C01810=1192.674,149.566,-54.225,-178.267,6.243,148.616
C01811=1192.678,149.317,-54.204,-178.270,6.241,148.616
C01812=1192.683,149.068,-54.182,-178.272,6.240,148.617
C01813=1192.688,148.819,-54.161,-178.275,6.239,148.617
C01814=1192.693,148.570,-54.141,-178.278,6.237,148.618
C01815=1192.698,148.321,-54.119,-178.281,6.235,148.618
C01816=1192.701,148.072,-54.099,-178.283,6.234,148.618
C01817=1192.707,147.823,-54.078,-178.286,6.232,148.619
C01818=1192.712,147.573,-54.057,-178.289,6.231,148.619
C01819=1192.716,147.324,-54.036,-178.291,6.229,148.620
C01820=1192.721,147.076,-54.015,-178.294,6.228,148.620
C01821=1192.726,146.827,-53.994,-178.296,6.226,148.620
C01822=1192.731,146.577,-53.973,-178.299,6.225,148.621
C01823=1192.735,146.329,-53.953,-178.302,6.223,148.621
C01824=1192.740,146.079,-53.932,-178.304,6.222,148.622
C01825=1192.744,145.830,-53.911,-178.307,6.221,148.622
C01826=1192.749,145.581,-53.890,-178.310,6.219,148.623
C01827=1192.753,145.332,-53.869,-178.312,6.217,148.623
C01828=1192.759,145.083,-53.848,-178.315,6.216,148.624
C01829=1192.763,144.834,-53.828,-178.318,6.215,148.624
C01830=1192.768,144.585,-53.807,-178.320,6.213,148.624
C01831=1192.773,144.336,-53.787,-178.323,6.211,148.625
C01832=1192.778,144.086,-53.766,-178.325,6.211,148.625
C01833=1192.782,143.837,-53.745,-178.328,6.209,148.626
C01834=1192.787,143.588,-53.724,-178.331,6.207,148.626
C01835=1192.792,143.339,-53.704,-178.334,6.205,148.627
C01836=1192.797,143.091,-53.682,-178.336,6.204,148.627
C01837=1192.801,142.842,-53.662,-178.339,6.203,148.628
C01838=1192.806,142.592,-53.641,-178.342,6.201,148.628
C01839=1192.811,142.343,-53.620,-178.344,6.200,148.628
C01840=1192.815,142.093,-53.599,-178.346,6.198,148.629
C01841=1192.820,141.844,-53.579,-178.349,6.197,148.629
C01842=1192.824,141.596,-53.558,-178.352,6.195,148.630
C01843=1192.830,141.346,-53.538,-178.354,6.194,148.630
C01844=1192.834,141.097,-53.518,-178.357,6.192,148.630
C01845=1192.839,140.847,-53.497,-178.360,6.191,148.631
C01846=1192.844,140.598,-53.476,-178.362,6.190,148.632
C01847=1192.848,140.350,-53.456,-178.365,6.188,148.632
C01848=1192.853,140.100,-53.435,-178.368,6.187,148.632
C01849=1192.858,139.851,-53.415,-178.371,6.185,148.633
C01850=1192.862,139.602,-53.394,-178.373,6.184,148.633
C01851=1192.867,139.353,-53.373,-178.376,6.182,148.634
C01852=1192.872,139.104,-53.353,-178.378,6.181,148.634
C01853=1192.877,138.856,-53.333,-178.381,6.180,148.635
C01854=1192.882,138.606,-53.313,-178.384,6.178,148.635
C01855=1192.887,138.357,-53.292,-178.386,6.176,148.635
C01856=1192.891,138.108,-53.272,-178.388,6.176,148.636
C01857=1192.896,137.859,-53.251,-178.392,6.174,148.636
C01858=1192.901,137.610,-53.231,-178.394,6.172,148.637
C01859=1192.905,137.361,-53.210,-178.397,6.171,148.637
C01860=1192.911,137.111,-53.190,-178.399,6.170,148.638
C01861=1192.915,136.862,-53.170,-178.402,6.168,148.638
C01862=1192.920,136.613,-53.149,-178.405,6.166,148.639
C01863=1192.924,136.364,-53.129,-178.407,6.165,148.639
C01864=1192.930,136.114,-53.109,-178.410,6.164,148.639
C01865=1192.934,135.865,-53.088,-178.413,6.162,148.640
C01866=1192.938,135.616,-53.068,-178.415,6.161,148.640
C01867=1192.943,135.368,-53.048,-178.418,6.160,148.641
C01868=1192.949,135.118,-53.028,-178.420,6.158,148.641
C01869=1192.953,134.869,-53.007,-178.423,6.157,148.642
C01870=1192.958,134.620,-52.987,-178.426,6.155,148.642
C01871=1192.963,134.371,-52.967,-178.428,6.154,148.643
C01872=1192.967,134.122,-52.947,-178.431,6.153,148.643
C01873=1192.972,133.873,-52.926,-178.434,6.151,148.644
C01874=1192.977,133.623,-52.906,-178.436,6.150,148.644
C01875=1192.981,133.374,-52.886,-178.438,6.149,148.644
C01876=1192.987,133.105,-52.864,-178.442,6.147,148.645
C01877=1192.992,132.837,-52.842,-178.444,6.145,148.645
C01878=1192.997,132.568,-52.821,-178.448,6.144,148.646
C01879=1193.002,132.300,-52.799,-178.450,6.142,148.646
C01880=1193.007,132.051,-52.779,-178.453,6.142,148.647
C01881=1193.011,131.802,-52.759,-178.456,6.140,148.647
C01882=1193.017,131.552,-52.739,-178.458,6.138,148.648
C01883=1193.022,131.304,-52.719,-178.461,6.138,148.648
C01884=1193.026,131.054,-52.699,-178.464,6.136,148.649
C01885=1193.031,130.805,-52.679,-178.466,6.134,148.649
C01886=1193.036,130.555,-52.659,-178.468,6.133,148.650
C01887=1193.040,130.307,-52.639,-178.472,6.132,148.650
C01888=1193.045,130.058,-52.619,-178.474,6.130,148.651
C01889=1193.050,129.809,-52.599,-178.476,6.129,148.651
C01890=1193.055,129.559,-52.579,-178.479,6.128,148.652
C01891=1193.060,129.310,-52.558,-178.482,6.126,148.652
C01892=1193.064,129.060,-52.539,-178.484,6.125,148.652
C01893=1193.069,128.812,-52.519,-178.487,6.123,148.653
C01894=1193.074,128.562,-52.499,-178.490,6.123,148.653
C01895=1193.079,128.314,-52.479,-178.492,6.121,148.654
C01896=1193.083,128.064,-52.459,-178.495,6.119,148.655
C01897=1193.088,127.816,-52.439,-178.498,6.118,148.655
C01898=1193.093,127.566,-52.419,-178.500,6.117,148.655
C01899=1193.098,127.317,-52.400,-178.503,6.115,148.656
C01900=1193.102,127.068,-52.379,-178.506,6.114,148.656
C01901=1193.108,126.819,-52.360,-178.508,6.113,148.657
C01902=1193.112,126.569,-52.340,-178.510,6.112,148.657
C01903=1193.117,126.320,-52.320,-178.514,6.110,148.658
C01904=1193.122,126.071,-52.300,-178.516,6.108,148.658
C01905=1193.127,125.822,-52.281,-178.518,6.107,148.659
C01906=1193.131,125.573,-52.261,-178.522,6.106,148.659
C01907=1193.136,125.323,-52.241,-178.524,6.105,148.660
C01908=1193.141,125.074,-52.221,-178.526,6.103,148.660
C01909=1193.146,124.825,-52.201,-178.530,6.102,148.661
C01910=1193.150,124.576,-52.182,-178.532,6.101,148.661
C01911=1193.155,124.327,-52.163,-178.534,6.099,148.661
C01912=1193.159,124.077,-52.143,-178.538,6.098,148.662
C01913=1193.164,123.829,-52.123,-178.540,6.097,148.662
C01914=1193.169,123.579,-52.103,-178.542,6.095,148.663
C01915=1193.174,123.330,-52.084,-178.545,6.095,148.663
C01916=1193.179,123.081,-52.064,-178.548,6.093,148.664
C01917=1193.184,122.832,-52.044,-178.550,6.092,148.664
C01918=1193.188,122.582,-52.024,-178.553,6.090,148.665
C01919=1193.194,122.333,-52.005,-178.556,6.089,148.665
C01920=1193.198,122.084,-51.986,-178.558,6.088,148.666
C01921=1193.203,121.835,-51.966,-178.561,6.086,148.666
C01922=1193.208,121.586,-51.946,-178.563,6.085,148.667
C01923=1193.212,121.337,-51.927,-178.566,6.084,148.667
C01924=1193.217,121.087,-51.907,-178.569,6.082,148.668
C01925=1193.222,120.838,-51.888,-178.571,6.081,148.668
C01926=1193.227,120.589,-51.868,-178.574,6.080,148.669
C01927=1193.231,120.340,-51.849,-178.576,6.079,148.669
C01928=1193.237,120.091,-51.830,-178.579,6.077,148.670
C01929=1193.241,119.841,-51.810,-178.582,6.076,148.670
C01930=1193.246,119.592,-51.790,-178.584,6.075,148.671
C01931=1193.251,119.343,-51.770,-178.588,6.074,148.671
C01932=1193.255,119.094,-51.751,-178.590,6.073,148.672
C01933=1193.260,118.845,-51.732,-178.592,6.071,148.672
C01934=1193.265,118.596,-51.712,-178.595,6.070,148.673
C01935=1193.270,118.346,-51.693,-178.598,6.068,148.673
C01936=1193.274,118.097,-51.674,-178.600,6.068,148.673
C01937=1193.279,117.848,-51.654,-178.603,6.066,148.674
C01938=1193.285,117.599,-51.635,-178.606,6.064,148.674
C01939=1193.289,117.349,-51.615,-178.608,6.064,148.675
C01940=1193.293,117.100,-51.596,-178.611,6.062,148.676
C01941=1193.299,116.851,-51.577,-178.613,6.061,148.676
C01942=1193.303,116.602,-51.557,-178.616,6.060,148.677
C01943=1193.309,116.353,-51.538,-178.618,6.059,148.677
C01944=1193.313,116.104,-51.519,-178.621,6.057,148.677
C01945=1193.318,115.854,-51.500,-178.624,6.056,148.678
C01946=1193.323,115.605,-51.481,-178.627,6.055,148.678
C01947=1193.328,115.356,-51.462,-178.630,6.053,148.679
C01948=1193.333,115.106,-51.442,-178.632,6.052,148.679
C01949=1193.337,114.857,-51.423,-178.635,6.051,148.680
C01950=1193.342,114.608,-51.404,-178.637,6.050,148.681
C01951=1193.347,114.359,-51.384,-178.640,6.048,148.681
C01952=1193.352,114.110,-51.365,-178.642,6.048,148.682
C01953=1193.356,113.861,-51.346,-178.645,6.046,148.682
C01954=1193.362,113.611,-51.328,-178.647,6.045,148.682
C01955=1193.366,113.362,-51.308,-178.650,6.044,148.683
C01956=1193.371,113.113,-51.289,-178.653,6.043,148.683
C01957=1193.376,112.863,-51.270,-178.656,6.041,148.684
C01958=1193.381,112.615,-51.250,-178.658,6.040,148.684
C01959=1193.385,112.365,-51.232,-178.661,6.039,148.685
C01960=1193.391,112.116,-51.213,-178.664,6.037,148.685
C01961=1193.395,111.867,-51.194,-178.666,6.036,148.686
C01962=1193.400,111.618,-51.174,-178.669,6.035,148.687
C01963=1193.405,111.368,-51.155,-178.671,6.034,148.687
C01964=1193.410,111.119,-51.137,-178.674,6.032,148.687
C01965=1193.414,110.869,-51.117,-178.677,6.032,148.688
C01966=1193.419,110.621,-51.098,-178.679,6.030,148.688
C01967=1193.424,110.371,-51.079,-178.682,6.029,148.689
C01968=1193.429,110.122,-51.061,-178.685,6.028,148.689
C01969=1193.434,109.873,-51.041,-178.687,6.027,148.690
C01970=1193.438,109.624,-51.022,-178.690,6.025,148.690
C01971=1193.444,109.375,-51.004,-178.692,6.024,148.691
C01972=1193.448,109.125,-50.985,-178.695,6.023,148.691
C01973=1193.453,108.876,-50.965,-178.697,6.022,148.692
C01974=1193.457,108.627,-50.947,-178.700,6.021,148.693
C01975=1193.463,108.378,-50.928,-178.703,6.020,148.693
C01976=1193.467,108.128,-50.909,-178.706,6.018,148.694
C01977=1193.472,107.879,-50.890,-178.708,6.017,148.694
C01978=1193.477,107.630,-50.871,-178.711,6.016,148.694
C01979=1193.482,107.380,-50.852,-178.713,6.015,148.695
C01980=1193.488,107.112,-50.832,-178.716,6.013,148.695
C01981=1193.492,106.843,-50.812,-178.719,6.012,148.696
C01982=1193.498,106.575,-50.791,-178.722,6.011,148.697
C01983=1193.503,106.307,-50.772,-178.724,6.010,148.697
C01984=1193.507,106.057,-50.752,-178.727,6.009,148.698
C01985=1193.512,105.808,-50.734,-178.730,6.007,148.698
C01986=1193.518,105.559,-50.715,-178.732,6.007,148.699
C01987=1193.522,105.310,-50.697,-178.735,6.005,148.699
C01988=1193.527,105.061,-50.677,-178.738,6.004,148.700
C01989=1193.532,104.811,-50.659,-178.740,6.003,148.700
C01990=1193.536,104.562,-50.640,-178.743,6.002,148.701
C01991=1193.542,104.313,-50.622,-178.746,6.000,148.701
C01992=1193.546,104.064,-50.603,-178.748,5.999,148.702
C01993=1193.551,103.814,-50.584,-178.751,5.998,148.702
C01994=1193.556,103.565,-50.565,-178.753,5.997,148.703
C01995=1193.560,103.316,-50.547,-178.756,5.996,148.703
C01996=1193.566,103.066,-50.528,-178.759,5.995,148.704
C01997=1193.571,102.818,-50.510,-178.762,5.993,148.704
C01998=1193.575,102.568,-50.491,-178.764,5.992,148.705
C01999=1193.580,102.319,-50.472,-178.767,5.991,148.706
C02000=1193.585,102.070,-50.454,-178.769,5.990,148.706
C02001=1193.590,101.820,-50.436,-178.771,5.989,148.706
C02002=1193.595,101.571,-50.416,-178.774,5.988,148.707
C02003=1193.600,101.322,-50.398,-178.777,5.987,148.707
C02004=1193.604,101.072,-50.379,-178.780,5.985,148.708
C02005=1193.609,100.823,-50.361,-178.782,5.985,148.708
C02006=1193.614,100.574,-50.343,-178.785,5.983,148.709
C02007=1193.619,100.325,-50.324,-178.787,5.982,148.710
C02008=1193.623,100.075,-50.306,-178.790,5.981,148.710
C02009=1193.629,99.826,-50.287,-178.793,5.980,148.711
C02010=1193.634,99.577,-50.269,-178.796,5.979,148.711
C02011=1193.638,99.327,-50.250,-178.798,5.978,148.712
C02012=1193.643,99.078,-50.232,-178.801,5.977,148.712
C02013=1193.648,98.829,-50.214,-178.803,5.975,148.713
C02014=1193.653,98.580,-50.195,-178.806,5.975,148.713
C02015=1193.657,98.330,-50.177,-178.809,5.973,148.714
C02016=1193.662,98.081,-50.159,-178.811,5.972,148.714
C02017=1193.668,97.832,-50.140,-178.814,5.971,148.715
C02018=1193.673,97.583,-50.122,-178.816,5.970,148.715
C02019=1193.677,97.333,-50.103,-178.819,5.968,148.716
C02020=1193.682,97.084,-50.085,-178.821,5.967,148.716
C02021=1193.687,96.835,-50.067,-178.824,5.967,148.717
C02022=1193.692,96.585,-50.048,-178.827,5.965,148.717
C02023=1193.697,96.336,-50.030,-178.829,5.965,148.718
C02024=1193.701,96.087,-50.011,-178.832,5.963,148.718
C02025=1193.706,95.838,-49.993,-178.835,5.962,148.719
C02026=1193.711,95.589,-49.975,-178.837,5.961,148.719
C02027=1193.716,95.339,-49.957,-178.840,5.960,148.720
C02028=1193.720,95.090,-49.939,-178.842,5.959,148.721
C02029=1193.726,94.840,-49.921,-178.845,5.958,148.721
C02030=1193.731,94.591,-49.903,-178.847,5.957,148.722
C02031=1193.736,94.342,-49.885,-178.851,5.955,148.722
C02032=1193.741,94.093,-49.867,-178.853,5.954,148.723
C02033=1193.745,93.843,-49.848,-178.855,5.954,148.723
C02034=1193.750,93.594,-49.830,-178.858,5.952,148.724
C02035=1193.754,93.345,-49.812,-178.861,5.952,148.724
C02036=1193.759,93.096,-49.794,-178.863,5.950,148.725
C02037=1193.764,92.847,-49.776,-178.866,5.949,148.725
C02038=1193.770,92.597,-49.757,-178.868,5.948,148.726
C02039=1193.774,92.347,-49.739,-178.871,5.947,148.727
C02040=1193.779,92.098,-49.721,-178.874,5.946,148.727
C02041=1193.784,91.849,-49.703,-178.877,5.945,148.728
C02042=1193.789,91.600,-49.685,-178.879,5.944,148.728
C02043=1193.794,91.351,-49.667,-178.881,5.943,148.729
C02044=1193.799,91.101,-49.649,-178.884,5.941,148.729
C02045=1193.804,90.852,-49.631,-178.887,5.941,148.730
C02046=1193.808,90.602,-49.613,-178.890,5.939,148.730
C02047=1193.813,90.353,-49.595,-178.892,5.939,148.731
C02048=1193.818,90.104,-49.577,-178.895,5.938,148.731
C02049=1193.823,89.854,-49.559,-178.897,5.936,148.732
C02050=1193.828,89.605,-49.541,-178.900,5.936,148.732
C02051=1193.833,89.356,-49.523,-178.903,5.934,148.733
C02052=1193.838,89.107,-49.505,-178.905,5.933,148.734
C02053=1193.843,88.857,-49.487,-178.908,5.933,148.734
C02054=1193.848,88.608,-49.469,-178.911,5.931,148.735
C02055=1193.852,88.358,-49.451,-178.913,5.930,148.735
C02056=1193.857,88.109,-49.433,-178.916,5.930,148.736
C02057=1193.862,87.859,-49.416,-178.918,5.928,148.736
C02058=1193.867,87.610,-49.398,-178.921,5.927,148.737
C02059=1193.872,87.361,-49.380,-178.924,5.926,148.737
C02060=1193.877,87.112,-49.362,-178.926,5.925,148.738
C02061=1193.882,86.863,-49.344,-178.928,5.924,148.738
C02062=1193.886,86.614,-49.326,-178.932,5.923,148.739
C02063=1193.891,86.364,-49.309,-178.934,5.922,148.739
C02064=1193.896,86.115,-49.291,-178.936,5.921,148.740
C02065=1193.901,85.866,-49.273,-178.939,5.920,148.741
C02066=1193.906,85.617,-49.255,-178.942,5.919,148.741
C02067=1193.911,85.367,-49.238,-178.945,5.918,148.742
C02068=1193.916,85.118,-49.220,-178.947,5.917,148.742
C02069=1193.921,84.868,-49.202,-178.950,5.916,148.743
C02070=1193.926,84.619,-49.184,-178.952,5.915,148.743
C02071=1193.930,84.370,-49.167,-178.955,5.914,148.744
C02072=1193.935,84.121,-49.149,-178.957,5.913,148.744
C02073=1193.940,83.871,-49.131,-178.960,5.912,148.745
C02074=1193.945,83.622,-49.114,-178.962,5.911,148.745
C02075=1193.950,83.372,-49.096,-178.965,5.910,148.746
C02076=1193.955,83.123,-49.078,-178.968,5.909,148.747
C02077=1193.960,82.874,-49.062,-178.970,5.908,148.747
C02078=1193.965,82.625,-49.044,-178.973,5.907,148.748
C02079=1193.969,82.375,-49.026,-178.976,5.906,148.748
C02080=1193.975,82.126,-49.008,-178.978,5.905,148.749
C02081=1193.980,81.876,-48.990,-178.980,5.904,148.749
C02082=1193.984,81.628,-48.973,-178.984,5.903,148.750
C02083=1193.989,81.378,-48.956,-178.986,5.902,148.750
C02084=1193.994,81.110,-48.936,-178.989,5.901,148.751
C02085=1193.999,80.841,-48.918,-178.992,5.900,148.752
C02086=1194.005,80.572,-48.898,-178.995,5.899,148.752
C02087=1194.010,80.304,-48.880,-178.997,5.898,148.753
C02088=1194.015,80.055,-48.862,-179.000,5.897,148.753
C02089=1194.020,79.806,-48.845,-179.003,5.896,148.754
C02090=1194.025,79.556,-48.827,-179.005,5.895,148.754
C02091=1194.030,79.307,-48.810,-179.008,5.894,148.755
C02092=1194.034,79.058,-48.793,-179.010,5.893,148.755
C02093=1194.039,78.808,-48.775,-179.013,5.892,148.756
C02094=1194.044,78.559,-48.757,-179.015,5.891,148.757
C02095=1194.050,78.309,-48.740,-179.018,5.890,148.757
C02096=1194.054,78.060,-48.723,-179.021,5.889,148.758
C02097=1194.059,77.810,-48.705,-179.023,5.888,148.758
C02098=1194.064,77.561,-48.687,-179.026,5.887,148.759
C02099=1194.068,77.312,-48.671,-179.028,5.886,148.759
C02100=1194.074,77.063,-48.653,-179.031,5.885,148.760
C02101=1194.079,76.813,-48.636,-179.034,5.884,148.760
C02102=1194.084,76.564,-48.619,-179.036,5.883,148.761
C02103=1194.088,76.315,-48.601,-179.039,5.883,148.762
C02104=1194.094,76.065,-48.584,-179.042,5.881,148.762
C02105=1194.098,75.816,-48.567,-179.044,5.880,148.763
C02106=1194.103,75.566,-48.549,-179.046,5.879,148.763
C02107=1194.108,75.317,-48.533,-179.049,5.879,148.764
C02108=1194.112,75.068,-48.515,-179.052,5.878,148.765
C02109=1194.118,74.819,-48.498,-179.054,5.877,148.765
C02110=1194.123,74.569,-48.481,-179.057,5.876,148.766
C02111=1194.128,74.320,-48.463,-179.060,5.874,148.766
C02112=1194.133,74.070,-48.446,-179.062,5.874,148.767
C02113=1194.137,73.821,-48.429,-179.065,5.873,148.767
C02114=1194.142,73.571,-48.411,-179.068,5.872,148.768
C02115=1194.147,73.323,-48.395,-179.070,5.871,148.769
C02116=1194.153,73.073,-48.378,-179.073,5.870,148.769
C02117=1194.157,72.824,-48.360,-179.075,5.870,148.770
C02118=1194.162,72.574,-48.343,-179.078,5.868,148.770
C02119=1194.166,72.325,-48.326,-179.080,5.867,148.771
C02120=1194.172,72.075,-48.309,-179.083,5.867,148.771
C02121=1194.177,71.826,-48.291,-179.085,5.866,148.772
C02122=1194.182,71.577,-48.275,-179.088,5.864,148.772
C02123=1194.187,71.327,-48.258,-179.091,5.864,148.773
C02124=1194.191,71.078,-48.241,-179.093,5.863,148.774
C02125=1194.196,70.828,-48.223,-179.096,5.862,148.774
C02126=1194.201,70.580,-48.207,-179.099,5.861,148.775
C02127=1194.207,70.330,-48.189,-179.101,5.860,148.775
C02128=1194.211,70.080,-48.173,-179.104,5.860,148.776
C02129=1194.216,69.831,-48.155,-179.107,5.858,148.776
C02130=1194.220,69.582,-48.138,-179.109,5.857,148.777
C02131=1194.226,69.333,-48.121,-179.111,5.856,148.777
C02132=1194.231,69.083,-48.104,-179.114,5.856,148.778
C02133=1194.236,68.833,-48.087,-179.117,5.855,148.779
C02134=1194.240,68.584,-48.071,-179.119,5.854,148.779
C02135=1194.246,68.335,-48.054,-179.122,5.853,148.780
C02136=1194.251,68.085,-48.037,-179.125,5.851,148.780
C02137=1194.255,67.836,-48.020,-179.127,5.851,148.781
C02138=1194.260,67.587,-48.002,-179.130,5.850,148.782
C02139=1194.265,67.338,-47.986,-179.132,5.849,148.782
C02140=1194.270,67.088,-47.969,-179.135,5.848,148.783
C02141=1194.275,66.839,-47.952,-179.138,5.848,148.783
C02142=1194.279,66.589,-47.935,-179.140,5.847,148.784
C02143=1194.285,66.340,-47.918,-179.143,5.846,148.784
C02144=1194.290,66.091,-47.902,-179.145,5.844,148.785
C02145=1194.295,65.841,-47.885,-179.148,5.844,148.786
C02146=1194.300,65.592,-47.868,-179.151,5.843,148.786
C02147=1194.304,65.342,-47.852,-179.153,5.842,148.787
C02148=1194.310,65.093,-47.834,-179.156,5.841,148.787
C02149=1194.314,64.843,-47.818,-179.159,5.840,148.788
C02150=1194.319,64.594,-47.801,-179.161,5.840,148.788
C02151=1194.324,64.345,-47.784,-179.163,5.839,148.789
C02152=1194.329,64.095,-47.767,-179.166,5.838,148.790
C02153=1194.334,63.846,-47.751,-179.169,5.837,148.790
C02154=1194.339,63.597,-47.734,-179.171,5.836,148.791
C02155=1194.344,63.347,-47.717,-179.174,5.835,148.791
C02156=1194.349,63.098,-47.701,-179.176,5.835,148.792
C02157=1194.354,62.848,-47.684,-179.179,5.833,148.793
C02158=1194.358,62.599,-47.667,-179.182,5.833,148.793
C02159=1194.364,62.350,-47.651,-179.184,5.832,148.794
C02160=1194.369,62.100,-47.634,-179.186,5.831,148.794
C02161=1194.374,61.850,-47.617,-179.190,5.830,148.795
C02162=1194.379,61.602,-47.601,-179.192,5.829,148.795
C02163=1194.383,61.352,-47.584,-179.194,5.828,148.796
C02164=1194.388,61.102,-47.567,-179.197,5.828,148.797
C02165=1194.393,60.853,-47.551,-179.200,5.827,148.797
C02166=1194.398,60.604,-47.534,-179.202,5.826,148.798
C02167=1194.403,60.355,-47.519,-179.205,5.825,148.798
C02168=1194.409,60.105,-47.501,-179.208,5.824,148.799
C02169=1194.413,59.855,-47.485,-179.210,5.824,148.799
C02170=1194.418,59.607,-47.468,-179.212,5.823,148.800
C02171=1194.423,59.357,-47.452,-179.216,5.822,148.801
C02172=1194.429,59.107,-47.436,-179.218,5.821,148.801
C02173=1194.433,58.858,-47.419,-179.220,5.820,148.802
C02174=1194.438,58.608,-47.402,-179.223,5.820,148.802
C02175=1194.443,58.360,-47.386,-179.225,5.819,148.803
C02176=1194.448,58.109,-47.370,-179.228,5.817,148.804
C02177=1194.453,57.860,-47.353,-179.231,5.817,148.804
C02178=1194.458,57.611,-47.336,-179.233,5.816,148.805
C02179=1194.462,57.361,-47.320,-179.236,5.815,148.805
C02180=1194.468,57.112,-47.304,-179.238,5.815,148.806
C02181=1194.472,56.863,-47.287,-179.241,5.813,148.806
C02182=1194.477,56.614,-47.271,-179.244,5.813,148.807
C02183=1194.483,56.363,-47.255,-179.246,5.812,148.808
C02184=1194.488,56.115,-47.238,-179.249,5.811,148.808
C02185=1194.492,55.865,-47.222,-179.251,5.811,148.809
C02186=1194.498,55.616,-47.206,-179.254,5.809,148.809
C02187=1194.502,55.366,-47.189,-179.257,5.809,148.810
C02188=1194.508,55.098,-47.172,-179.259,5.808,148.811
C02189=1194.512,54.829,-47.154,-179.262,5.807,148.811
C02190=1194.519,54.560,-47.137,-179.265,5.806,148.812
C02191=1194.524,54.292,-47.119,-179.268,5.806,148.813
C02192=1194.529,54.042,-47.103,-179.270,5.805,148.813
C02193=1194.534,53.794,-47.087,-179.273,5.803,148.814
C02194=1194.538,53.544,-47.070,-179.276,5.803,148.814
C02195=1194.544,53.295,-47.054,-179.278,5.802,148.815
C02196=1194.548,53.045,-47.038,-179.280,5.801,148.816
C02197=1194.554,52.796,-47.022,-179.283,5.801,148.816
C02198=1194.558,52.546,-47.005,-179.285,5.800,148.817
C02199=1194.563,52.297,-46.990,-179.288,5.799,148.817
C02200=1194.568,52.047,-46.973,-179.291,5.798,148.818
C02201=1194.573,51.798,-46.958,-179.293,5.797,148.818
C02202=1194.578,51.549,-46.941,-179.296,5.797,148.819
C02203=1194.583,51.299,-46.925,-179.299,5.796,148.820
C02204=1194.588,51.050,-46.909,-179.301,5.795,148.820
C02205=1194.593,50.800,-46.893,-179.304,5.794,148.821
C02206=1194.597,50.551,-46.876,-179.307,5.793,148.822
C02207=1194.603,50.301,-46.861,-179.309,5.792,148.822
C02208=1194.607,50.052,-46.844,-179.311,5.792,148.823
C02209=1194.613,49.803,-46.829,-179.314,5.791,148.823
C02210=1194.617,49.553,-46.812,-179.316,5.791,148.824
C02211=1194.623,49.304,-46.796,-179.319,5.789,148.824
C02212=1194.628,49.055,-46.780,-179.322,5.789,148.825
C02213=1194.632,48.805,-46.764,-179.324,5.788,148.826
C02214=1194.638,48.555,-46.748,-179.327,5.787,148.826
C02215=1194.642,48.306,-46.732,-179.329,5.787,148.827
C02216=1194.648,48.056,-46.716,-179.332,5.786,148.827
C02217=1194.652,47.807,-46.700,-179.334,5.785,148.828
C02218=1194.658,47.558,-46.684,-179.337,5.784,148.829
C02219=1194.663,47.308,-46.668,-179.340,5.783,148.829
C02220=1194.667,47.059,-46.652,-179.342,5.783,148.830
C02221=1194.673,46.809,-46.636,-179.345,5.782,148.830
C02222=1194.678,46.559,-46.620,-179.347,5.781,148.831
C02223=1194.683,46.310,-46.604,-179.350,5.781,148.832
C02224=1194.687,46.061,-46.589,-179.352,5.780,148.832
C02225=1194.692,45.811,-46.573,-179.355,5.779,148.833
C02226=1194.697,45.562,-46.557,-179.358,5.778,148.833
C02227=1194.702,45.312,-46.541,-179.360,5.777,148.834
C02228=1194.707,45.063,-46.525,-179.363,5.777,148.835
C02229=1194.712,44.814,-46.509,-179.366,5.776,148.835
C02230=1194.717,44.564,-46.493,-179.368,5.775,148.836
C02231=1194.723,44.315,-46.477,-179.370,5.775,148.836
C02232=1194.727,44.066,-46.462,-179.373,5.774,148.837
C02233=1194.732,43.816,-46.446,-179.376,5.773,148.838
C02234=1194.737,43.567,-46.430,-179.378,5.772,148.838
C02235=1194.742,43.317,-46.414,-179.381,5.772,148.839
C02236=1194.747,43.067,-46.398,-179.383,5.771,148.839
C02237=1194.753,42.818,-46.383,-179.386,5.770,148.840
C02238=1194.756,42.569,-46.367,-179.388,5.770,148.841
C02239=1194.762,42.319,-46.351,-179.391,5.769,148.841
C02240=1194.767,42.070,-46.336,-179.393,5.768,148.842
C02241=1194.773,41.820,-46.320,-179.396,5.768,148.842
C02242=1194.777,41.570,-46.304,-179.399,5.766,148.843
C02243=1194.782,41.322,-46.288,-179.401,5.766,148.844
C02244=1194.787,41.072,-46.273,-179.404,5.765,148.844
C02245=1194.792,40.822,-46.257,-179.407,5.764,148.845
C02246=1194.797,40.573,-46.241,-179.409,5.764,148.845
C02247=1194.802,40.324,-46.226,-179.411,5.763,148.846
C02248=1194.807,40.074,-46.210,-179.414,5.763,148.847
C02249=1194.812,39.824,-46.195,-179.417,5.762,148.847
C02250=1194.818,39.575,-46.179,-179.419,5.761,148.848
C02251=1194.822,39.326,-46.164,-179.422,5.760,148.849
C02252=1194.827,39.076,-46.147,-179.425,5.759,148.849
C02253=1194.832,38.827,-46.132,-179.427,5.758,148.850
C02254=1194.837,38.577,-46.116,-179.429,5.758,148.850
C02255=1194.841,38.328,-46.101,-179.432,5.757,148.851
C02256=1194.847,38.078,-46.085,-179.435,5.757,148.852
C02257=1194.852,37.829,-46.070,-179.437,5.756,148.852
C02258=1194.857,37.580,-46.055,-179.439,5.755,148.853
C02259=1194.862,37.330,-46.039,-179.442,5.755,148.853
C02260=1194.867,37.080,-46.023,-179.445,5.754,148.854
C02261=1194.872,36.831,-46.008,-179.447,5.754,148.855
C02262=1194.877,36.582,-45.993,-179.450,5.752,148.855
C02263=1194.882,36.332,-45.977,-179.453,5.752,148.856
C02264=1194.887,36.083,-45.962,-179.455,5.751,148.856
C02265=1194.892,35.833,-45.946,-179.458,5.750,148.857
C02266=1194.897,35.584,-45.930,-179.460,5.750,148.858
C02267=1194.902,35.335,-45.915,-179.463,5.749,148.858
C02268=1194.907,35.085,-45.900,-179.465,5.748,148.859
C02269=1194.912,34.835,-45.884,-179.468,5.748,148.860
C02270=1194.917,34.585,-45.870,-179.470,5.747,148.860
C02271=1194.922,34.336,-45.854,-179.472,5.746,148.861
C02272=1194.927,34.087,-45.839,-179.475,5.746,148.861
C02273=1194.932,33.837,-45.823,-179.478,5.745,148.862
C02274=1194.937,33.587,-45.808,-179.480,5.745,148.863
C02275=1194.942,33.338,-45.793,-179.483,5.744,148.863
C02276=1194.947,33.089,-45.777,-179.486,5.743,148.864
C02277=1194.952,32.840,-45.762,-179.488,5.742,148.864
C02278=1194.957,32.590,-45.746,-179.491,5.742,148.865
C02279=1194.962,32.340,-45.732,-179.493,5.741,148.866
C02280=1194.967,32.091,-45.716,-179.496,5.740,148.866
C02281=1194.972,31.842,-45.701,-179.499,5.740,148.867
C02282=1194.977,31.592,-45.686,-179.501,5.739,148.868
C02283=1194.983,31.343,-45.670,-179.503,5.738,148.868
C02284=1194.987,31.093,-45.655,-179.506,5.738,148.869
C02285=1194.992,30.843,-45.640,-179.509,5.737,148.869
C02286=1194.997,30.594,-45.625,-179.511,5.736,148.870
C02287=1195.002,30.344,-45.609,-179.513,5.736,148.871
C02288=1195.007,30.095,-45.594,-179.516,5.735,148.871
C02289=1195.013,29.845,-45.579,-179.519,5.735,148.872
C02290=1195.017,29.596,-45.564,-179.521,5.734,148.872
C02291=1195.022,29.346,-45.548,-179.523,5.734,148.873
C02292=1195.027,29.077,-45.533,-179.527,5.732,148.874
C02293=1195.033,28.809,-45.516,-179.529,5.732,148.874
C02294=1195.038,28.540,-45.500,-179.532,5.731,148.875
C02295=1195.044,28.271,-45.484,-179.535,5.731,148.876
C02296=1195.048,28.022,-45.469,-179.537,5.730,148.876
C02297=1195.054,27.773,-45.453,-179.539,5.729,148.877
C02298=1195.059,27.523,-45.439,-179.542,5.729,148.878
C02299=1195.064,27.273,-45.423,-179.545,5.728,148.878
C02300=1195.069,27.024,-45.408,-179.547,5.728,148.879
C02301=1195.074,26.775,-45.394,-179.550,5.727,148.879
C02302=1195.079,26.525,-45.378,-179.552,5.726,148.880
C02303=1195.084,26.276,-45.363,-179.555,5.726,148.881
C02304=1195.089,26.026,-45.348,-179.557,5.725,148.881
C02305=1195.094,25.776,-45.333,-179.560,5.725,148.882
C02306=1195.099,25.527,-45.318,-179.563,5.723,148.883
C02307=1195.104,25.277,-45.303,-179.566,5.723,148.883
C02308=1195.109,25.028,-45.288,-179.568,5.722,148.884
C02309=1195.114,24.778,-45.273,-179.570,5.721,148.884
C02310=1195.119,24.529,-45.258,-179.573,5.721,148.885
C02311=1195.124,24.279,-45.244,-179.576,5.720,148.886
C02312=1195.129,24.030,-45.229,-179.578,5.720,148.886
C02313=1195.134,23.781,-45.214,-179.580,5.719,148.887
C02314=1195.139,23.531,-45.199,-179.583,5.718,148.888
C02315=1195.144,23.282,-45.184,-179.586,5.718,148.888
C02316=1195.149,23.032,-45.169,-179.588,5.717,148.889
C02317=1195.154,22.783,-45.154,-179.591,5.717,148.889
C02318=1195.160,22.533,-45.140,-179.593,5.716,148.890
C02319=1195.164,22.284,-45.125,-179.596,5.715,148.891
C02320=1195.169,22.034,-45.110,-179.598,5.715,148.891
C02321=1195.174,21.785,-45.095,-179.601,5.714,148.892
C02322=1195.179,21.535,-45.080,-179.603,5.714,148.892
C02323=1195.184,21.286,-45.065,-179.606,5.713,148.893
C02324=1195.190,21.036,-45.051,-179.609,5.713,148.894
C02325=1195.194,20.787,-45.036,-179.611,5.712,148.895
C02326=1195.199,20.537,-45.021,-179.613,5.711,148.895
C02327=1195.205,20.288,-45.006,-179.616,5.711,148.896
C02328=1195.210,20.038,-44.991,-179.619,5.710,148.896
C02329=1195.215,19.788,-44.977,-179.621,5.710,148.897
C02330=1195.219,19.539,-44.962,-179.623,5.709,148.897
C02331=1195.225,19.289,-44.947,-179.626,5.708,148.898
C02332=1195.230,19.040,-44.932,-179.629,5.708,148.899
C02333=1195.235,18.790,-44.918,-179.631,5.707,148.900
C02334=1195.240,18.541,-44.904,-179.634,5.706,148.900
C02335=1195.244,18.291,-44.889,-179.636,5.706,148.901
C02336=1195.250,18.041,-44.874,-179.639,5.705,148.901
C02337=1195.255,17.792,-44.860,-179.642,5.705,148.902
C02338=1195.260,17.543,-44.845,-179.644,5.704,148.902
C02339=1195.264,17.293,-44.830,-179.646,5.704,148.903
C02340=1195.270,17.043,-44.815,-179.649,5.703,148.904
C02341=1195.275,16.794,-44.800,-179.652,5.703,148.905
C02342=1195.280,16.545,-44.787,-179.654,5.702,148.905
C02343=1195.285,16.295,-44.772,-179.656,5.701,148.906
C02344=1195.290,16.046,-44.757,-179.659,5.701,148.906
C02345=1195.295,15.796,-44.743,-179.662,5.700,148.907
C02346=1195.301,15.546,-44.728,-179.664,5.700,148.908
C02347=1195.305,15.297,-44.713,-179.667,5.699,148.908
C02348=1195.310,15.047,-44.699,-179.669,5.699,148.909
C02349=1195.315,14.798,-44.685,-179.671,5.699,148.910
C02350=1195.320,14.548,-44.670,-179.674,5.698,148.910
C02351=1195.325,14.299,-44.655,-179.677,5.698,148.911
C02352=1195.330,14.050,-44.641,-179.679,5.697,148.911
C02353=1195.336,13.800,-44.626,-179.681,5.696,148.912
C02354=1195.341,13.550,-44.612,-179.684,5.696,148.913
C02355=1195.346,13.301,-44.598,-179.687,5.695,148.913
C02356=1195.351,13.051,-44.583,-179.689,5.694,148.914
C02357=1195.356,12.802,-44.569,-179.691,5.694,148.915
C02358=1195.361,12.552,-44.554,-179.694,5.693,148.915
C02359=1195.365,12.302,-44.540,-179.697,5.693,148.916
C02360=1195.371,12.053,-44.526,-179.699,5.692,148.916
C02361=1195.376,11.804,-44.512,-179.702,5.692,148.917
C02362=1195.381,11.554,-44.497,-179.704,5.691,148.918
C02363=1195.386,11.305,-44.483,-179.707,5.691,148.918
C02364=1195.391,11.055,-44.468,-179.710,5.690,148.919
C02365=1195.396,10.805,-44.453,-179.712,5.689,148.920
C02366=1195.401,10.555,-44.439,-179.714,5.689,148.920
C02367=1195.407,10.306,-44.425,-179.717,5.688,148.921
C02368=1195.412,10.057,-44.411,-179.720,5.688,148.922
C02369=1195.417,9.807,-44.397,-179.722,5.687,148.922
C02370=1195.421,9.558,-44.382,-179.724,5.686,148.923
C02371=1195.426,9.308,-44.367,-179.727,5.686,148.923
C02372=1195.432,9.059,-44.354,-179.729,5.686,148.924
C02373=1195.437,8.809,-44.339,-179.732,5.686,148.925
C02374=1195.442,8.560,-44.325,-179.734,5.685,148.925
C02375=1195.447,8.310,-44.311,-179.737,5.684,148.926
C02376=1195.452,8.060,-44.296,-179.739,5.684,148.927
C02377=1195.457,7.811,-44.283,-179.742,5.683,148.927
C02378=1195.462,7.562,-44.268,-179.745,5.683,148.928
C02379=1195.467,7.312,-44.254,-179.747,5.682,148.928
C02380=1195.472,7.062,-44.240,-179.749,5.681,148.929
C02381=1195.477,6.812,-44.225,-179.752,5.681,148.930
C02382=1195.483,6.563,-44.212,-179.755,5.681,148.931
C02383=1195.488,6.314,-44.197,-179.757,5.680,148.931
C02384=1195.492,6.064,-44.184,-179.760,5.679,148.932
C02385=1195.497,5.815,-44.169,-179.762,5.679,148.932
C02386=1195.502,5.566,-44.155,-179.765,5.678,148.933
C02387=1195.507,5.316,-44.141,-179.767,5.678,148.934
C02388=1195.512,5.066,-44.127,-179.769,5.678,148.934
C02389=1195.517,4.816,-44.113,-179.772,5.677,148.935
C02390=1195.523,4.567,-44.099,-179.774,5.677,148.936
C02391=1195.528,4.317,-44.085,-179.777,5.676,148.936
C02392=1195.533,4.067,-44.071,-179.780,5.676,148.937
C02393=1195.538,3.818,-44.057,-179.782,5.675,148.937
C02394=1195.543,3.569,-44.043,-179.785,5.674,148.938
C02395=1195.548,3.319,-44.029,-179.787,5.674,148.939
C02396=1195.553,3.050,-44.014,-179.790,5.673,148.939
C02397=1195.558,2.780,-43.999,-179.792,5.673,148.940
C02398=1195.564,2.512,-43.983,-179.795,5.672,148.941
C02399=1195.570,2.243,-43.969,-179.798,5.672,148.942
C02400=1195.575,1.993,-43.954,-179.800,5.671,148.942
C02401=1195.580,1.743,-43.940,-179.803,5.671,148.943
C02402=1195.585,1.494,-43.927,-179.805,5.670,148.943
C02403=1195.590,1.244,-43.913,-179.808,5.670,148.944
C02404=1195.595,0.994,-43.898,-179.811,5.669,148.945
C02405=1195.600,0.745,-43.885,-179.813,5.669,148.945
C02406=1195.605,0.496,-43.871,-179.815,5.669,148.946
C02407=1195.610,0.246,-43.857,-179.817,5.668,148.947
C02408=1195.615,-0.004,-43.843,-179.820,5.668,148.947
C02409=1195.621,-0.253,-43.829,-179.823,5.667,148.948
C02410=1195.625,-0.502,-43.815,-179.825,5.667,148.949
C02411=1195.630,-0.753,-43.802,-179.828,5.666,148.949
C02412=1195.636,-1.002,-43.788,-179.830,5.665,148.950
C02413=1195.641,-1.251,-43.774,-179.833,5.665,148.950
C02414=1195.646,-1.500,-43.760,-179.836,5.664,148.951
C02415=1195.651,-1.750,-43.747,-179.838,5.664,148.952
C02416=1195.656,-2.000,-43.732,-179.840,5.664,148.952
C02417=1195.661,-2.249,-43.718,-179.842,5.663,148.953
C02418=1195.667,-2.500,-43.705,-179.845,5.663,148.954
C02419=1195.671,-2.749,-43.691,-179.848,5.662,148.954
C02420=1195.676,-2.998,-43.677,-179.850,5.662,148.955
C02421=1195.682,-3.248,-43.664,-179.853,5.661,148.956
C02422=1195.687,-3.498,-43.649,-179.855,5.660,148.956
C02423=1195.692,-3.747,-43.636,-179.858,5.660,148.957
C02424=1195.697,-3.997,-43.623,-179.861,5.659,148.958
C02425=1195.702,-4.246,-43.609,-179.863,5.660,148.958
C02426=1195.707,-4.495,-43.595,-179.865,5.659,148.959
C02427=1195.712,-4.746,-43.581,-179.867,5.658,148.959
C02428=1195.717,-4.995,-43.568,-179.870,5.658,148.960
C02429=1195.722,-5.245,-43.555,-179.873,5.657,148.961
C02430=1195.727,-5.494,-43.541,-179.875,5.657,148.962
C02431=1195.732,-5.744,-43.526,-179.878,5.656,148.962
C02432=1195.737,-5.994,-43.513,-179.880,5.656,148.963
C02433=1195.742,-6.243,-43.500,-179.882,5.656,148.963
C02434=1195.748,-6.493,-43.486,-179.885,5.656,148.964
C02435=1195.753,-6.742,-43.473,-179.888,5.655,148.965
C02436=1195.758,-6.992,-43.459,-179.890,5.654,148.965
C02437=1195.763,-7.241,-43.445,-179.892,5.654,148.966
C02438=1195.768,-7.490,-43.431,-179.895,5.653,148.967
C02439=1195.773,-7.741,-43.418,-179.898,5.653,148.967
C02440=1195.778,-7.990,-43.404,-179.900,5.653,148.968
C02441=1195.783,-8.240,-43.391,-179.902,5.653,148.969
C02442=1195.788,-8.489,-43.377,-179.905,5.652,148.969
C02443=1195.793,-8.739,-43.364,-179.907,5.651,148.970
C02444=1195.799,-8.988,-43.350,-179.910,5.651,148.971
C02445=1195.804,-9.238,-43.337,-179.913,5.650,148.971
C02446=1195.809,-9.487,-43.323,-179.915,5.650,148.972
C02447=1195.814,-9.737,-43.310,-179.917,5.650,148.972
C02448=1195.819,-9.986,-43.297,-179.920,5.649,148.973
C02449=1195.824,-10.236,-43.283,-179.922,5.649,148.974
C02450=1195.828,-10.486,-43.270,-179.925,5.648,148.974
C02451=1195.834,-10.735,-43.256,-179.927,5.648,148.975
C02452=1195.839,-10.985,-43.242,-179.930,5.647,148.976
C02453=1195.844,-11.234,-43.229,-179.932,5.647,148.976
C02454=1195.849,-11.484,-43.216,-179.934,5.647,148.977
C02455=1195.855,-11.734,-43.203,-179.937,5.646,148.978
C02456=1195.859,-11.984,-43.189,-179.940,5.646,148.978
C02457=1195.865,-12.233,-43.176,-179.942,5.645,148.979
C02458=1195.870,-12.483,-43.162,-179.945,5.645,148.980
C02459=1195.875,-12.732,-43.149,-179.947,5.644,148.980
C02460=1195.880,-12.982,-43.136,-179.950,5.644,148.981
C02461=1195.885,-13.231,-43.122,-179.952,5.644,148.982
C02462=1195.891,-13.480,-43.109,-179.954,5.643,148.982
C02463=1195.895,-13.731,-43.096,-179.957,5.643,148.983
C02464=1195.901,-13.980,-43.082,-179.959,5.642,148.983
C02465=1195.905,-14.230,-43.069,-179.962,5.642,148.984
C02466=1195.911,-14.479,-43.056,-179.965,5.641,148.985
C02467=1195.915,-14.729,-43.042,-179.966,5.641,148.985
C02468=1195.921,-14.978,-43.029,-179.969,5.641,148.986
C02469=1195.926,-15.228,-43.016,-179.972,5.640,148.987
C02470=1195.932,-15.478,-43.003,-179.974,5.640,148.987
C02471=1195.936,-15.727,-42.989,-179.977,5.639,148.988
C02472=1195.941,-15.977,-42.977,-179.979,5.638,148.989
C02473=1195.947,-16.226,-42.964,-179.981,5.639,148.989
C02474=1195.951,-16.476,-42.951,-179.984,5.638,148.990
C02475=1195.957,-16.725,-42.937,-179.986,5.638,148.991
C02476=1195.961,-16.975,-42.924,-179.989,5.637,148.991
C02477=1195.967,-17.225,-42.911,-179.992,5.637,148.992
C02478=1195.972,-17.475,-42.898,-179.993,5.637,148.992
C02479=1195.977,-17.724,-42.884,-179.996,5.636,148.993
C02480=1195.982,-17.973,-42.871,-179.999,5.636,148.994
C02481=1195.987,-18.223,-42.858,179.999,5.635,148.995
C02482=1195.993,-18.473,-42.845,179.996,5.635,148.995
C02483=1195.997,-18.723,-42.832,179.994,5.634,148.996
C02484=1196.002,-18.972,-42.819,179.992,5.634,148.996
C02485=1196.008,-19.221,-42.805,179.989,5.634,148.997
C02486=1196.013,-19.471,-42.792,179.986,5.633,148.998
C02487=1196.018,-19.721,-42.780,179.984,5.633,148.999
C02488=1196.023,-19.970,-42.767,179.982,5.632,148.999
C02489=1196.028,-20.220,-42.754,179.980,5.632,149.000
C02490=1196.034,-20.470,-42.741,179.977,5.632,149.000
C02491=1196.038,-20.720,-42.728,179.974,5.632,149.001
C02492=1196.043,-20.969,-42.714,179.972,5.631,149.002
C02493=1196.049,-21.218,-42.701,179.969,5.630,149.002
C02494=1196.054,-21.468,-42.688,179.967,5.631,149.003
C02495=1196.059,-21.718,-42.675,179.965,5.630,149.004
C02496=1196.065,-21.967,-42.662,179.962,5.630,149.004
C02497=1196.069,-22.217,-42.649,179.959,5.629,149.005
C02498=1196.074,-22.466,-42.637,179.957,5.629,149.006
C02499=1196.079,-22.716,-42.624,179.955,5.629,149.006
C02500=1196.085,-22.986,-42.610,179.952,5.628,149.007
C02501=1196.090,-23.256,-42.596,179.950,5.628,149.008
C02502=1196.096,-23.525,-42.582,179.947,5.627,149.008
C02503=1196.101,-23.795,-42.569,179.944,5.627,149.009
C02504=1196.107,-24.044,-42.555,179.942,5.626,149.010
C02505=1196.112,-24.294,-42.542,179.939,5.626,149.010
C02506=1196.117,-24.544,-42.530,179.936,5.625,149.011
C02507=1196.122,-24.793,-42.517,179.934,5.626,149.012
C02508=1196.127,-25.043,-42.504,179.932,5.625,149.012
C02509=1196.132,-25.293,-42.491,179.930,5.624,149.013
C02510=1196.138,-25.542,-42.478,179.927,5.624,149.014
C02511=1196.143,-25.791,-42.466,179.924,5.623,149.014
C02512=1196.148,-26.042,-42.452,179.922,5.624,149.015
C02513=1196.153,-26.291,-42.440,179.919,5.623,149.016
C02514=1196.158,-26.540,-42.427,179.917,5.623,149.016
C02515=1196.163,-26.790,-42.414,179.915,5.622,149.017
C02516=1196.168,-27.039,-42.402,179.913,5.622,149.018
C02517=1196.174,-27.289,-42.388,179.910,5.622,149.018
C02518=1196.179,-27.538,-42.376,179.907,5.621,149.019
C02519=1196.183,-27.788,-42.363,179.905,5.621,149.019
C02520=1196.188,-28.038,-42.350,179.902,5.620,149.020
C02521=1196.194,-28.287,-42.338,179.900,5.620,149.021
C02522=1196.199,-28.537,-42.326,179.898,5.620,149.021
C02523=1196.204,-28.787,-42.312,179.895,5.620,149.022
C02524=1196.209,-29.037,-42.300,179.892,5.619,149.023
C02525=1196.215,-29.286,-42.287,179.891,5.619,149.023
C02526=1196.220,-29.535,-42.274,179.888,5.619,149.024
C02527=1196.224,-29.785,-42.261,179.885,5.618,149.025
C02528=1196.229,-30.035,-42.249,179.883,5.618,149.025
C02529=1196.235,-30.285,-42.237,179.880,5.617,149.026
C02530=1196.241,-30.534,-42.224,179.879,5.617,149.027
C02531=1196.245,-30.784,-42.211,179.876,5.617,149.027
C02532=1196.250,-31.034,-42.198,179.873,5.616,149.028
C02533=1196.255,-31.283,-42.185,179.871,5.616,149.029
C02534=1196.261,-31.533,-42.174,179.868,5.616,149.029
C02535=1196.266,-31.782,-42.161,179.866,5.615,149.030
C02536=1196.270,-32.032,-42.148,179.864,5.615,149.031
C02537=1196.276,-32.281,-42.135,179.861,5.614,149.031
C02538=1196.281,-32.531,-42.124,179.859,5.615,149.032
C02539=1196.286,-32.781,-42.111,179.856,5.614,149.033
C02540=1196.292,-33.030,-42.098,179.854,5.614,149.033
C02541=1196.297,-33.280,-42.085,179.851,5.613,149.034
C02542=1196.302,-33.530,-42.073,179.849,5.613,149.035
C02543=1196.307,-33.780,-42.060,179.847,5.613,149.035
C02544=1196.312,-34.029,-42.048,179.844,5.612,149.036
C02545=1196.318,-34.279,-42.036,179.841,5.612,149.037
C02546=1196.323,-34.528,-42.023,179.840,5.612,149.037
C02547=1196.327,-34.778,-42.010,179.837,5.611,149.038
C02548=1196.333,-35.028,-41.998,179.834,5.611,149.039
C02549=1196.338,-35.277,-41.986,179.832,5.611,149.039
C02550=1196.343,-35.527,-41.973,179.830,5.611,149.040
C02551=1196.348,-35.777,-41.961,179.827,5.610,149.040
C02552=1196.354,-36.026,-41.949,179.825,5.610,149.041
C02553=1196.359,-36.275,-41.936,179.822,5.609,149.042
C02554=1196.363,-36.526,-41.924,179.820,5.609,149.042
C02555=1196.369,-36.775,-41.911,179.817,5.609,149.043
C02556=1196.374,-37.025,-41.899,179.815,5.608,149.044
C02557=1196.379,-37.275,-41.887,179.813,5.608,149.044
C02558=1196.384,-37.524,-41.874,179.810,5.608,149.045
C02559=1196.390,-37.774,-41.862,179.808,5.608,149.046
C02560=1196.395,-38.023,-41.850,179.805,5.607,149.046
C02561=1196.400,-38.272,-41.837,179.802,5.607,149.047
C02562=1196.405,-38.523,-41.825,179.801,5.607,149.048
C02563=1196.410,-38.772,-41.812,179.798,5.606,149.048
C02564=1196.415,-39.022,-41.800,179.796,5.606,149.049
C02565=1196.420,-39.272,-41.788,179.793,5.606,149.050
C02566=1196.426,-39.522,-41.776,179.791,5.606,149.050
C02567=1196.430,-39.771,-41.764,179.789,5.605,149.051
C02568=1196.436,-40.021,-41.752,179.786,5.604,149.052
C02569=1196.441,-40.270,-41.739,179.784,5.605,149.052
C02570=1196.446,-40.520,-41.727,179.781,5.604,149.053
C02571=1196.451,-40.769,-41.715,179.779,5.604,149.054
C02572=1196.457,-41.019,-41.703,179.776,5.603,149.054
C02573=1196.462,-41.268,-41.690,179.774,5.603,149.055
C02574=1196.467,-41.519,-41.678,179.772,5.603,149.056
C02575=1196.472,-41.768,-41.666,179.769,5.602,149.056
C02576=1196.477,-42.018,-41.654,179.767,5.603,149.057
C02577=1196.482,-42.267,-41.642,179.765,5.602,149.057
C02578=1196.487,-42.517,-41.630,179.762,5.601,149.058
C02579=1196.492,-42.767,-41.617,179.759,5.601,149.059
C02580=1196.498,-43.016,-41.605,179.757,5.601,149.060
C02581=1196.503,-43.266,-41.593,179.755,5.601,149.060
C02582=1196.508,-43.516,-41.581,179.752,5.600,149.061
C02583=1196.513,-43.765,-41.569,179.750,5.600,149.061
C02584=1196.518,-44.015,-41.557,179.748,5.600,149.062
C02585=1196.523,-44.265,-41.545,179.745,5.600,149.063
C02586=1196.529,-44.514,-41.532,179.742,5.599,149.064
C02587=1196.534,-44.764,-41.520,179.741,5.599,149.064
C02588=1196.539,-45.014,-41.509,179.738,5.599,149.065
C02589=1196.544,-45.263,-41.497,179.735,5.598,149.065
C02590=1196.549,-45.513,-41.485,179.733,5.599,149.066
C02591=1196.555,-45.763,-41.473,179.731,5.598,149.067
C02592=1196.560,-46.012,-41.460,179.729,5.597,149.067
C02593=1196.565,-46.262,-41.448,179.726,5.597,149.068
C02594=1196.570,-46.512,-41.437,179.724,5.597,149.069
C02595=1196.575,-46.761,-41.424,179.721,5.597,149.069
C02596=1196.580,-47.011,-41.413,179.718,5.596,149.070
C02597=1196.586,-47.261,-41.401,179.717,5.596,149.071
C02598=1196.590,-47.510,-41.389,179.714,5.596,149.071
C02599=1196.596,-47.760,-41.377,179.712,5.595,149.072
C02600=1196.601,-48.010,-41.365,179.710,5.596,149.073
C02601=1196.606,-48.259,-41.352,179.707,5.595,149.073
C02602=1196.611,-48.509,-41.341,179.705,5.594,149.074
C02603=1196.616,-48.758,-41.329,179.702,5.594,149.075
C02604=1196.622,-49.028,-41.317,179.700,5.594,149.075
C02605=1196.628,-49.298,-41.304,179.697,5.594,149.076
C02606=1196.633,-49.569,-41.291,179.695,5.593,149.077
C02607=1196.640,-49.839,-41.277,179.692,5.593,149.077
C02608=1196.644,-50.088,-41.266,179.689,5.593,149.078
C02609=1196.650,-50.338,-41.254,179.687,5.593,149.079
C02610=1196.655,-50.588,-41.242,179.684,5.592,149.079
C02611=1196.660,-50.837,-41.230,179.682,5.592,149.080
C02612=1196.665,-51.087,-41.218,179.680,5.592,149.081
C02613=1196.670,-51.337,-41.207,179.678,5.592,149.081
C02614=1196.675,-51.587,-41.195,179.675,5.591,149.082
C02615=1196.680,-51.836,-41.183,179.673,5.591,149.083
C02616=1196.686,-52.086,-41.171,179.670,5.591,149.083
C02617=1196.690,-52.336,-41.160,179.668,5.590,149.084
C02618=1196.696,-52.586,-41.148,179.666,5.591,149.085
C02619=1196.702,-52.835,-41.136,179.663,5.590,149.085
C02620=1196.706,-53.084,-41.125,179.661,5.590,149.086
C02621=1196.712,-53.334,-41.113,179.658,5.590,149.087
C02622=1196.717,-53.584,-41.100,179.656,5.589,149.087
C02623=1196.722,-53.833,-41.089,179.654,5.589,149.088
C02624=1196.727,-54.083,-41.077,179.652,5.589,149.089
C02625=1196.732,-54.333,-41.066,179.649,5.589,149.089
C02626=1196.737,-54.583,-41.054,179.646,5.588,149.090
C02627=1196.743,-54.833,-41.042,179.645,5.588,149.091
C02628=1196.747,-55.082,-41.031,179.642,5.588,149.091
C02629=1196.753,-55.332,-41.019,179.639,5.587,149.092
C02630=1196.758,-55.581,-41.008,179.637,5.588,149.093
C02631=1196.764,-55.831,-40.996,179.635,5.587,149.093
C02632=1196.768,-56.081,-40.985,179.632,5.586,149.094
C02633=1196.774,-56.331,-40.973,179.630,5.587,149.095
C02634=1196.779,-56.580,-40.960,179.628,5.586,149.095
C02635=1196.783,-56.830,-40.949,179.625,5.586,149.096
C02636=1196.790,-57.079,-40.938,179.623,5.586,149.096
C02637=1196.794,-57.329,-40.926,179.621,5.585,149.097
C02638=1196.800,-57.579,-40.914,179.618,5.585,149.098
C02639=1196.804,-57.828,-40.903,179.616,5.585,149.099
C02640=1196.810,-58.078,-40.891,179.613,5.585,149.099
C02641=1196.814,-58.328,-40.880,179.611,5.584,149.100
C02642=1196.820,-58.577,-40.868,179.609,5.584,149.100
C02643=1196.825,-58.827,-40.857,179.606,5.584,149.101
C02644=1196.831,-59.076,-40.845,179.604,5.584,149.102
C02645=1196.836,-59.327,-40.835,179.602,5.584,149.103
C02646=1196.841,-59.577,-40.823,179.599,5.583,149.103
C02647=1196.846,-59.826,-40.811,179.597,5.583,149.104
C02648=1196.852,-60.076,-40.800,179.595,5.583,149.104
C02649=1196.856,-60.325,-40.789,179.592,5.583,149.105
C02650=1196.862,-60.575,-40.777,179.590,5.582,149.106
C02651=1196.867,-60.825,-40.765,179.588,5.582,149.106
C02652=1196.872,-61.075,-40.754,179.585,5.582,149.107
C02653=1196.877,-61.324,-40.743,179.582,5.581,149.108
C02654=1196.883,-61.574,-40.731,179.580,5.582,149.108
C02655=1196.887,-61.823,-40.719,179.578,5.581,149.109
C02656=1196.893,-62.073,-40.708,179.575,5.580,149.110
C02657=1196.898,-62.323,-40.697,179.573,5.581,149.110
C02658=1196.904,-62.573,-40.685,179.571,5.580,149.111
C02659=1196.909,-62.822,-40.674,179.569,5.579,149.111
C02660=1196.913,-63.072,-40.663,179.566,5.580,149.112
C02661=1196.919,-63.322,-40.651,179.564,5.579,149.113
C02662=1196.924,-63.571,-40.640,179.562,5.580,149.114
C02663=1196.930,-63.821,-40.629,179.559,5.579,149.114
C02664=1196.934,-64.071,-40.618,179.557,5.579,149.115
C02665=1196.939,-64.320,-40.606,179.555,5.579,149.115
C02666=1196.945,-64.570,-40.595,179.552,5.578,149.116
C02667=1196.950,-64.819,-40.584,179.549,5.578,149.117
C02668=1196.955,-65.069,-40.572,179.548,5.578,149.117
C02669=1196.960,-65.320,-40.561,179.545,5.578,149.118
C02670=1196.966,-65.568,-40.550,179.542,5.577,149.119
C02671=1196.971,-65.818,-40.538,179.540,5.577,149.119
C02672=1196.976,-66.068,-40.527,179.538,5.577,149.120
C02673=1196.982,-66.318,-40.516,179.536,5.577,149.121
C02674=1196.987,-66.568,-40.505,179.533,5.577,149.121
C02675=1196.991,-66.817,-40.494,179.531,5.576,149.122
C02676=1196.997,-67.067,-40.482,179.529,5.577,149.123
C02677=1197.002,-67.317,-40.472,179.527,5.576,149.123
C02678=1197.007,-67.566,-40.460,179.524,5.575,149.124
C02679=1197.013,-67.816,-40.448,179.522,5.576,149.125
C02680=1197.018,-68.066,-40.438,179.519,5.575,149.125
C02681=1197.023,-68.315,-40.427,179.517,5.576,149.126
C02682=1197.028,-68.565,-40.415,179.515,5.575,149.127
C02683=1197.034,-68.814,-40.404,179.512,5.574,149.127
C02684=1197.039,-69.064,-40.393,179.510,5.575,149.128
C02685=1197.044,-69.314,-40.382,179.507,5.574,149.129
C02686=1197.049,-69.563,-40.371,179.505,5.573,149.129
C02687=1197.054,-69.814,-40.360,179.503,5.574,149.130
C02688=1197.059,-70.063,-40.349,179.500,5.573,149.131
C02689=1197.065,-70.313,-40.338,179.498,5.574,149.131
C02690=1197.070,-70.563,-40.327,179.496,5.573,149.132
C02691=1197.075,-70.812,-40.315,179.494,5.573,149.132
C02692=1197.081,-71.062,-40.305,179.491,5.573,149.133
C02693=1197.086,-71.312,-40.293,179.489,5.572,149.134
C02694=1197.090,-71.561,-40.282,179.486,5.572,149.135
C02695=1197.096,-71.811,-40.272,179.485,5.572,149.135
C02696=1197.101,-72.061,-40.260,179.482,5.572,149.136
C02697=1197.106,-72.311,-40.249,179.480,5.572,149.136
C02698=1197.112,-72.560,-40.238,179.477,5.572,149.137
C02699=1197.116,-72.810,-40.227,179.475,5.571,149.138
C02700=1197.123,-73.060,-40.216,179.473,5.571,149.138
C02701=1197.127,-73.309,-40.205,179.470,5.571,149.139
C02702=1197.132,-73.559,-40.194,179.468,5.571,149.140
C02703=1197.138,-73.808,-40.184,179.466,5.570,149.140
C02704=1197.143,-74.059,-40.172,179.463,5.570,149.141
C02705=1197.149,-74.308,-40.161,179.461,5.570,149.142
C02706=1197.154,-74.558,-40.151,179.458,5.570,149.142
C02707=1197.158,-74.808,-40.140,179.457,5.570,149.143
C02708=1197.165,-75.078,-40.128,179.454,5.569,149.144
C02709=1197.171,-75.350,-40.116,179.452,5.569,149.144
C02710=1197.175,-75.620,-40.104,179.449,5.568,149.145
C02711=1197.182,-75.890,-40.093,179.447,5.569,149.146
C02712=1197.187,-76.141,-40.082,179.444,5.568,149.146
C02713=1197.192,-76.390,-40.071,179.441,5.568,149.147
C02714=1197.198,-76.640,-40.060,179.439,5.568,149.148
C02715=1197.203,-76.889,-40.049,179.437,5.568,149.148
C02716=1197.208,-77.139,-40.038,179.435,5.568,149.149
C02717=1197.213,-77.389,-40.027,179.432,5.568,149.150
C02718=1197.218,-77.639,-40.017,179.430,5.567,149.150
C02719=1197.223,-77.888,-40.006,179.428,5.567,149.151
C02720=1197.229,-78.138,-39.995,179.425,5.567,149.152
C02721=1197.234,-78.388,-39.984,179.423,5.567,149.152
C02722=1197.240,-78.637,-39.973,179.421,5.567,149.153
C02723=1197.245,-78.887,-39.963,179.419,5.566,149.154
C02724=1197.250,-79.136,-39.952,179.416,5.566,149.154
C02725=1197.255,-79.387,-39.941,179.414,5.566,149.155
C02726=1197.260,-79.637,-39.931,179.412,5.566,149.156
C02727=1197.265,-79.886,-39.920,179.410,5.565,149.156
C02728=1197.270,-80.136,-39.909,179.407,5.566,149.157
C02729=1197.275,-80.385,-39.898,179.405,5.565,149.158
C02730=1197.280,-80.635,-39.888,179.402,5.565,149.158
C02731=1197.287,-80.885,-39.877,179.400,5.565,149.159
C02732=1197.291,-81.135,-39.866,179.398,5.564,149.159
C02733=1197.297,-81.384,-39.855,179.396,5.565,149.160
C02734=1197.302,-81.634,-39.845,179.393,5.564,149.161
C02735=1197.307,-81.883,-39.834,179.391,5.564,149.161
C02736=1197.312,-82.134,-39.823,179.389,5.564,149.162
C02737=1197.318,-82.383,-39.813,179.386,5.564,149.163
C02738=1197.323,-82.633,-39.803,179.385,5.564,149.163
C02739=1197.328,-82.882,-39.792,179.382,5.563,149.164
C02740=1197.333,-83.133,-39.781,179.380,5.563,149.165
C02741=1197.339,-83.382,-39.771,179.377,5.563,149.165
C02742=1197.344,-83.632,-39.760,179.375,5.562,149.166
C02743=1197.349,-83.881,-39.749,179.373,5.563,149.167
C02744=1197.354,-84.132,-39.739,179.370,5.562,149.167
C02745=1197.360,-84.381,-39.729,179.368,5.563,149.168
C02746=1197.364,-84.631,-39.717,179.366,5.562,149.168
C02747=1197.370,-84.880,-39.707,179.364,5.562,149.169
C02748=1197.375,-85.131,-39.696,179.361,5.562,149.170
C02749=1197.381,-85.380,-39.686,179.358,5.561,149.171
C02750=1197.386,-85.630,-39.676,179.357,5.561,149.171
C02751=1197.391,-85.879,-39.665,179.354,5.561,149.172
C02752=1197.397,-86.129,-39.655,179.352,5.561,149.173
C02753=1197.402,-86.379,-39.644,179.350,5.560,149.173
C02754=1197.407,-86.629,-39.634,179.348,5.561,149.174
C02755=1197.412,-86.879,-39.623,179.345,5.560,149.174
C02756=1197.417,-87.128,-39.612,179.342,5.560,149.175
C02757=1197.422,-87.378,-39.602,179.341,5.560,149.176
C02758=1197.427,-87.627,-39.592,179.338,5.560,149.176
C02759=1197.433,-87.877,-39.582,179.336,5.560,149.177
C02760=1197.438,-88.127,-39.571,179.333,5.560,149.178
C02761=1197.443,-88.377,-39.561,179.332,5.560,149.178
C02762=1197.448,-88.626,-39.550,179.329,5.559,149.179
C02763=1197.454,-88.876,-39.540,179.327,5.560,149.180
C02764=1197.459,-89.126,-39.529,179.325,5.559,149.180
C02765=1197.464,-89.375,-39.519,179.322,5.558,149.181
C02766=1197.470,-89.625,-39.509,179.320,5.559,149.182
C02767=1197.475,-89.875,-39.498,179.317,5.558,149.182
C02768=1197.481,-90.125,-39.488,179.316,5.558,149.183
C02769=1197.485,-90.375,-39.478,179.313,5.558,149.183
C02770=1197.490,-90.624,-39.468,179.311,5.558,149.184
C02771=1197.496,-90.874,-39.457,179.309,5.557,149.185
C02772=1197.501,-91.124,-39.447,179.306,5.557,149.185
C02773=1197.506,-91.373,-39.436,179.304,5.557,149.186
C02774=1197.512,-91.623,-39.426,179.301,5.557,149.187
C02775=1197.517,-91.873,-39.415,179.300,5.557,149.187
C02776=1197.522,-92.122,-39.406,179.297,5.557,149.188
C02777=1197.527,-92.372,-39.395,179.295,5.557,149.189
C02778=1197.532,-92.622,-39.385,179.293,5.556,149.189
C02779=1197.538,-92.871,-39.375,179.291,5.557,149.190
C02780=1197.543,-93.122,-39.364,179.288,5.556,149.191
C02781=1197.549,-93.371,-39.354,179.287,5.556,149.191
C02782=1197.553,-93.620,-39.344,179.284,5.556,149.192
C02783=1197.558,-93.871,-39.334,179.281,5.555,149.193
C02784=1197.564,-94.120,-39.323,179.279,5.556,149.193
C02785=1197.570,-94.370,-39.313,179.277,5.555,149.194
C02786=1197.575,-94.620,-39.303,179.275,5.555,149.194
C02787=1197.579,-94.869,-39.293,179.272,5.555,149.195
C02788=1197.585,-95.119,-39.283,179.271,5.555,149.196
C02789=1197.590,-95.370,-39.273,179.268,5.554,149.196
C02790=1197.596,-95.619,-39.263,179.266,5.555,149.197
C02791=1197.602,-95.869,-39.252,179.263,5.554,149.198
C02792=1197.606,-96.119,-39.243,179.262,5.554,149.198
C02793=1197.611,-96.368,-39.232,179.259,5.554,149.199
C02794=1197.617,-96.618,-39.222,179.256,5.554,149.200
C02795=1197.622,-96.868,-39.212,179.255,5.554,149.200
C02796=1197.627,-97.117,-39.202,179.252,5.553,149.201
C02797=1197.632,-97.367,-39.192,179.250,5.554,149.202
C02798=1197.638,-97.616,-39.181,179.248,5.553,149.202
C02799=1197.643,-97.867,-39.171,179.246,5.553,149.203
C02800=1197.648,-98.116,-39.162,179.243,5.553,149.203
C02801=1197.654,-98.366,-39.152,179.241,5.553,149.204
C02802=1197.659,-98.616,-39.141,179.239,5.552,149.205
C02803=1197.664,-98.866,-39.131,179.237,5.553,149.205
C02804=1197.669,-99.115,-39.121,179.234,5.552,149.206
C02805=1197.675,-99.364,-39.111,179.232,5.552,149.207
C02806=1197.680,-99.615,-39.101,179.230,5.552,149.207
C02807=1197.685,-99.865,-39.092,179.228,5.552,149.208
C02808=1197.691,-100.114,-39.082,179.225,5.552,149.208
C02809=1197.696,-100.364,-39.071,179.223,5.552,149.209
C02810=1197.700,-100.614,-39.061,179.221,5.551,149.210
C02811=1197.706,-100.863,-39.051,179.218,5.551,149.210
C02812=1197.712,-101.135,-39.040,179.216,5.551,149.211
C02813=1197.718,-101.406,-39.030,179.214,5.551,149.212
C02814=1197.723,-101.677,-39.019,179.211,5.550,149.213
C02815=1197.730,-101.949,-39.008,179.209,5.551,149.213
C02816=1197.734,-102.199,-38.998,179.206,5.550,149.214
C02817=1197.740,-102.448,-38.988,179.205,5.550,149.214
C02818=1197.745,-102.699,-38.979,179.202,5.550,149.215
C02819=1197.750,-102.948,-38.969,179.200,5.550,149.216
C02820=1197.756,-103.198,-38.958,179.198,5.549,149.216
C02821=1197.761,-103.447,-38.949,179.196,5.550,149.217
C02822=1197.766,-103.698,-38.939,179.193,5.549,149.218
C02823=1197.771,-103.948,-38.929,179.191,5.549,149.218
C02824=1197.776,-104.197,-38.919,179.189,5.549,149.219
C02825=1197.782,-104.446,-38.909,179.186,5.549,149.220
C02826=1197.787,-104.696,-38.900,179.184,5.549,149.220
C02827=1197.792,-104.946,-38.889,179.182,5.549,149.221
C02828=1197.798,-105.196,-38.879,179.180,5.549,149.222
C02829=1197.803,-105.446,-38.870,179.178,5.549,149.222
C02830=1197.808,-105.695,-38.860,179.175,5.548,149.223
C02831=1197.813,-105.945,-38.851,179.173,5.549,149.224
C02832=1197.819,-106.195,-38.841,179.171,5.548,149.224
C02833=1197.824,-106.445,-38.831,179.169,5.548,149.225
C02834=1197.829,-106.694,-38.821,179.166,5.548,149.225
C02835=1197.835,-106.944,-38.811,179.165,5.548,149.226
C02836=1197.840,-107.194,-38.802,179.162,5.547,149.227
C02837=1197.846,-107.444,-38.792,179.159,5.547,149.227
C02838=1197.850,-107.694,-38.782,179.158,5.547,149.228
C02839=1197.856,-107.943,-38.772,179.155,5.547,149.229
C02840=1197.861,-108.193,-38.763,179.153,5.547,149.229
C02841=1197.866,-108.443,-38.753,179.151,5.546,149.230
C02842=1197.871,-108.692,-38.743,179.149,5.547,149.230
C02843=1197.877,-108.942,-38.734,179.146,5.546,149.231
C02844=1197.881,-109.192,-38.724,179.144,5.546,149.232
C02845=1197.887,-109.442,-38.714,179.142,5.546,149.232
C02846=1197.892,-109.691,-38.705,179.140,5.546,149.233
C02847=1197.898,-109.942,-38.695,179.137,5.545,149.234
C02848=1197.903,-110.191,-38.686,179.135,5.546,149.234
C02849=1197.909,-110.441,-38.676,179.133,5.545,149.235
C02850=1197.914,-110.690,-38.667,179.131,5.545,149.235
C02851=1197.919,-110.940,-38.656,179.128,5.545,149.236
C02852=1197.924,-111.190,-38.647,179.127,5.545,149.237
C02853=1197.929,-111.440,-38.637,179.124,5.545,149.237
C02854=1197.935,-111.690,-38.628,179.122,5.545,149.238
C02855=1197.940,-111.939,-38.618,179.120,5.544,149.239
C02856=1197.945,-112.189,-38.609,179.118,5.545,149.239
C02857=1197.951,-112.439,-38.599,179.115,5.544,149.240
C02858=1197.956,-112.688,-38.590,179.113,5.544,149.240
C02859=1197.962,-112.938,-38.580,179.111,5.544,149.241
C02860=1197.967,-113.188,-38.571,179.109,5.544,149.242
C02861=1197.973,-113.438,-38.561,179.106,5.543,149.242
C02862=1197.977,-113.688,-38.551,179.104,5.544,149.243
C02863=1197.982,-113.938,-38.542,179.102,5.543,149.244
C02864=1197.988,-114.187,-38.532,179.100,5.543,149.244
C02865=1197.993,-114.437,-38.523,179.097,5.543,149.245
C02866=1197.999,-114.687,-38.513,179.096,5.543,149.246
C02867=1198.004,-114.937,-38.504,179.094,5.543,149.246
C02868=1198.009,-115.186,-38.494,179.092,5.543,149.247
C02869=1198.015,-115.436,-38.485,179.089,5.543,149.247
C02870=1198.020,-115.686,-38.476,179.087,5.543,149.248
C02871=1198.025,-115.935,-38.466,179.085,5.543,149.249
C02872=1198.030,-116.185,-38.457,179.083,5.542,149.249
C02873=1198.035,-116.434,-38.447,179.080,5.543,149.250
C02874=1198.041,-116.685,-38.438,179.078,5.542,149.251
C02875=1198.046,-116.934,-38.429,179.076,5.542,149.251
C02876=1198.052,-117.184,-38.419,179.074,5.542,149.252
C02877=1198.057,-117.434,-38.410,179.072,5.542,149.252
C02878=1198.062,-117.684,-38.401,179.069,5.542,149.253
C02879=1198.068,-117.933,-38.391,179.068,5.542,149.254
C02880=1198.073,-118.184,-38.381,179.065,5.541,149.254
C02881=1198.078,-118.434,-38.373,179.063,5.541,149.255
C02882=1198.083,-118.683,-38.362,179.061,5.541,149.256
C02883=1198.088,-118.933,-38.353,179.059,5.541,149.256
C02884=1198.094,-119.183,-38.345,179.056,5.540,149.257
C02885=1198.099,-119.432,-38.334,179.054,5.541,149.258
C02886=1198.104,-119.682,-38.325,179.052,5.540,149.258
C02887=1198.110,-119.932,-38.317,179.050,5.540,149.259
C02888=1198.115,-120.182,-38.306,179.047,5.540,149.259
C02889=1198.120,-120.432,-38.297,179.046,5.540,149.260
C02890=1198.125,-120.681,-38.289,179.043,5.540,149.261
C02891=1198.131,-120.931,-38.280,179.041,5.540,149.261
C02892=1198.136,-121.181,-38.269,179.039,5.539,149.262
C02893=1198.141,-121.431,-38.261,179.037,5.540,149.263
C02894=1198.147,-121.680,-38.252,179.034,5.539,149.263
C02895=1198.152,-121.931,-38.242,179.032,5.539,149.264
C02896=1198.157,-122.180,-38.233,179.031,5.539,149.264
C02897=1198.163,-122.430,-38.224,179.028,5.539,149.265
C02898=1198.168,-122.680,-38.215,179.026,5.539,149.266
C02899=1198.174,-122.930,-38.205,179.024,5.538,149.266
C02900=1198.179,-123.178,-38.196,179.022,5.539,149.267
C02901=1198.184,-123.428,-38.187,179.020,5.538,149.267
C02902=1198.189,-123.678,-38.178,179.017,5.539,149.268
C02903=1198.195,-123.928,-38.169,179.015,5.538,149.269
C02904=1198.200,-124.178,-38.160,179.013,5.538,149.269
C02905=1198.206,-124.428,-38.151,179.010,5.538,149.270
C02906=1198.210,-124.677,-38.141,179.009,5.538,149.270
C02907=1198.216,-124.927,-38.132,179.006,5.537,149.271
C02908=1198.222,-125.177,-38.123,179.004,5.538,149.272
C02909=1198.227,-125.427,-38.114,179.002,5.537,149.272
C02910=1198.232,-125.677,-38.105,179.000,5.537,149.273
C02911=1198.237,-125.927,-38.096,178.998,5.537,149.274
C02912=1198.243,-126.176,-38.086,178.996,5.537,149.274
C02913=1198.248,-126.426,-38.077,178.994,5.537,149.275
C02914=1198.253,-126.676,-38.068,178.991,5.537,149.276
C02915=1198.258,-126.926,-38.059,178.989,5.537,149.276
C02916=1197.837,-126.937,-38.098,178.985,5.540,149.278
C02917=1197.832,-126.687,-38.107,178.987,5.540,149.277
C02918=1197.827,-126.437,-38.116,178.990,5.541,149.277
C02919=1197.821,-126.187,-38.125,178.992,5.540,149.276
C02920=1197.815,-125.937,-38.134,178.994,5.541,149.276
C02921=1197.810,-125.687,-38.143,178.996,5.541,149.275
C02922=1197.805,-125.438,-38.153,178.999,5.541,149.274
C02923=1197.800,-125.188,-38.162,179.000,5.541,149.274
C02924=1197.795,-124.938,-38.171,179.002,5.541,149.273
C02925=1197.789,-124.688,-38.180,179.004,5.541,149.273
C02926=1197.784,-124.438,-38.189,179.007,5.541,149.272
C02927=1197.779,-124.188,-38.198,179.009,5.541,149.271
C02928=1197.774,-123.939,-38.208,179.011,5.541,149.271
C02929=1197.767,-123.690,-38.217,179.014,5.542,149.270
C02930=1197.762,-123.440,-38.226,179.015,5.542,149.269
C02931=1197.757,-123.190,-38.234,179.018,5.542,149.269
C02932=1197.752,-122.940,-38.243,179.019,5.542,149.268
C02933=1197.746,-122.691,-38.254,179.022,5.542,149.268
C02934=1197.741,-122.441,-38.262,179.024,5.542,149.267
C02935=1197.736,-122.191,-38.271,179.026,5.543,149.266
C02936=1197.731,-121.941,-38.280,179.028,5.542,149.266
C02937=1197.725,-121.691,-38.290,179.031,5.543,149.265
C02938=1197.720,-121.442,-38.299,179.033,5.543,149.264
C02939=1197.715,-121.192,-38.308,179.035,5.543,149.264
C02940=1197.710,-120.942,-38.317,179.037,5.543,149.263
C02941=1197.704,-120.692,-38.327,179.039,5.543,149.263
C02942=1197.699,-120.442,-38.336,179.041,5.544,149.262
C02943=1197.694,-120.193,-38.345,179.043,5.543,149.261
C02944=1197.688,-119.942,-38.355,179.046,5.544,149.261
C02945=1197.683,-119.693,-38.364,179.048,5.544,149.260
C02946=1197.678,-119.443,-38.373,179.050,5.544,149.259
C02947=1197.672,-119.193,-38.383,179.052,5.544,149.259
C02948=1197.667,-118.944,-38.392,179.055,5.544,149.258
C02949=1197.662,-118.694,-38.401,179.057,5.544,149.257
C02950=1197.656,-118.444,-38.411,179.059,5.545,149.257
C02951=1197.651,-118.195,-38.420,179.061,5.544,149.256
C02952=1197.646,-117.945,-38.429,179.063,5.545,149.256
C02953=1197.640,-117.695,-38.439,179.065,5.545,149.255
C02954=1197.635,-117.446,-38.448,179.068,5.545,149.254
C02955=1197.630,-117.196,-38.457,179.070,5.545,149.254
C02956=1197.624,-116.945,-38.467,179.072,5.545,149.253
C02957=1197.620,-116.696,-38.477,179.074,5.545,149.253
C02958=1197.615,-116.446,-38.486,179.077,5.546,149.252
C02959=1197.609,-116.196,-38.495,179.079,5.545,149.251
C02960=1197.604,-115.946,-38.505,179.081,5.546,149.251
C02961=1197.598,-115.696,-38.514,179.083,5.546,149.250
C02962=1197.593,-115.447,-38.524,179.086,5.546,149.249
C02963=1197.588,-115.197,-38.533,179.087,5.546,149.249
C02964=1197.582,-114.947,-38.542,179.090,5.547,149.248
C02965=1197.577,-114.698,-38.552,179.091,5.547,149.248
C02966=1197.571,-114.448,-38.561,179.094,5.547,149.247
C02967=1197.567,-114.198,-38.571,179.096,5.547,149.246
C02968=1197.561,-113.948,-38.580,179.098,5.547,149.246
C02969=1197.556,-113.699,-38.590,179.100,5.547,149.245
C02970=1197.551,-113.449,-38.599,179.103,5.547,149.244
C02971=1197.545,-113.199,-38.608,179.105,5.547,149.244
C02972=1197.540,-112.950,-38.618,179.107,5.548,149.243
C02973=1197.535,-112.699,-38.628,179.109,5.548,149.243
C02974=1197.530,-112.450,-38.637,179.112,5.548,149.242
C02975=1197.525,-112.200,-38.646,179.114,5.548,149.241
C02976=1197.519,-111.950,-38.657,179.116,5.549,149.241
C02977=1197.514,-111.700,-38.665,179.118,5.548,149.240
C02978=1197.508,-111.451,-38.676,179.121,5.549,149.239
C02979=1197.503,-111.201,-38.685,179.122,5.549,149.239
C02980=1197.497,-110.951,-38.695,179.125,5.549,149.238
C02981=1197.492,-110.702,-38.704,179.127,5.549,149.238
C02982=1197.487,-110.451,-38.714,179.129,5.549,149.237
C02983=1197.482,-110.201,-38.723,179.131,5.549,149.236
C02984=1197.477,-109.952,-38.733,179.134,5.550,149.236
C02985=1197.472,-109.703,-38.743,179.136,5.549,149.235
C02986=1197.466,-109.452,-38.752,179.138,5.550,149.234
C02987=1197.461,-109.203,-38.762,179.140,5.550,149.234
C02988=1197.455,-108.953,-38.772,179.143,5.550,149.233
C02989=1197.450,-108.704,-38.781,179.145,5.550,149.232
C02990=1197.445,-108.453,-38.791,179.147,5.551,149.232
C02991=1197.440,-108.204,-38.801,179.149,5.550,149.231
C02992=1197.434,-107.954,-38.811,179.152,5.551,149.230
C02993=1197.429,-107.704,-38.820,179.153,5.551,149.230
C02994=1197.424,-107.455,-38.830,179.156,5.551,149.229
C02995=1197.418,-107.205,-38.839,179.158,5.551,149.228
C02996=1197.413,-106.955,-38.849,179.160,5.551,149.228
C02997=1197.408,-106.705,-38.860,179.162,5.551,149.227
C02998=1197.403,-106.455,-38.869,179.164,5.552,149.227
C02999=1197.397,-106.206,-38.879,179.167,5.551,149.226
C03000=1197.392,-105.957,-38.888,179.169,5.552,149.225
C03001=1197.386,-105.706,-38.898,179.171,5.552,149.225
C03002=1197.382,-105.456,-38.908,179.174,5.552,149.224
C03003=1197.376,-105.207,-38.918,179.176,5.552,149.223
C03004=1197.371,-104.957,-38.928,179.178,5.553,149.223
C03005=1197.366,-104.708,-38.937,179.180,5.552,149.222
C03006=1197.360,-104.458,-38.947,179.183,5.553,149.222
C03007=1197.356,-104.207,-38.957,179.184,5.553,149.221
C03008=1197.350,-103.958,-38.967,179.187,5.553,149.220
C03009=1197.344,-103.708,-38.977,179.189,5.553,149.220
C03010=1197.339,-103.459,-38.987,179.191,5.553,149.219
C03011=1197.334,-103.208,-38.996,179.193,5.553,149.218
C03012=1197.329,-102.959,-39.006,179.196,5.553,149.218
C03013=1197.324,-102.709,-39.016,179.197,5.553,149.217
C03014=1197.318,-102.459,-39.026,179.200,5.554,149.217
C03015=1197.313,-102.210,-39.035,179.202,5.553,149.216
C03016=1197.308,-101.960,-39.046,179.204,5.554,149.215
C03017=1197.302,-101.689,-39.057,179.207,5.555,149.215
C03018=1197.296,-101.417,-39.067,179.209,5.554,149.214
C03019=1197.291,-101.146,-39.078,179.212,5.555,149.213
C03020=1197.286,-100.874,-39.089,179.215,5.555,149.212
C03021=1197.280,-100.624,-39.099,179.217,5.555,149.212
C03022=1197.274,-100.375,-39.109,179.219,5.555,149.211
C03023=1197.269,-100.125,-39.119,179.221,5.555,149.211
C03024=1197.264,-99.875,-39.129,179.224,5.555,149.210
C03025=1197.259,-99.626,-39.139,179.225,5.555,149.209
C03026=1197.253,-99.376,-39.149,179.228,5.556,149.209
C03027=1197.248,-99.126,-39.159,179.230,5.555,149.208
C03028=1197.243,-98.876,-39.169,179.233,5.556,149.207
C03029=1197.237,-98.626,-39.179,179.234,5.556,149.207
C03030=1197.232,-98.377,-39.189,179.237,5.556,149.206
C03031=1197.227,-98.127,-39.199,179.239,5.556,149.205
C03032=1197.221,-97.877,-39.209,179.241,5.557,149.205
C03033=1197.216,-97.627,-39.219,179.243,5.556,149.204
C03034=1197.211,-97.378,-39.229,179.246,5.557,149.203
C03035=1197.206,-97.128,-39.239,179.248,5.558,149.203
C03036=1197.200,-96.878,-39.250,179.250,5.557,149.202
C03037=1197.195,-96.629,-39.260,179.253,5.558,149.201
C03038=1197.191,-96.379,-39.270,179.254,5.558,149.201
C03039=1197.185,-96.129,-39.280,179.257,5.558,149.200
C03040=1197.179,-95.880,-39.290,179.259,5.558,149.200
C03041=1197.174,-95.629,-39.301,179.261,5.558,149.199
C03042=1197.169,-95.380,-39.310,179.264,5.558,149.198
C03043=1197.164,-95.130,-39.320,179.266,5.558,149.198
C03044=1197.159,-94.880,-39.330,179.268,5.558,149.197
C03045=1197.153,-94.630,-39.341,179.270,5.559,149.196
C03046=1197.147,-94.381,-39.351,179.273,5.559,149.196
C03047=1197.143,-94.131,-39.361,179.275,5.559,149.195
C03048=1197.138,-93.881,-39.371,179.277,5.560,149.195
C03049=1197.132,-93.632,-39.381,179.279,5.559,149.194
C03050=1197.127,-93.381,-39.392,179.282,5.560,149.193
C03051=1197.121,-93.132,-39.402,179.284,5.560,149.193
C03052=1197.116,-92.882,-39.412,179.286,5.560,149.192
C03053=1197.111,-92.632,-39.422,179.289,5.560,149.191
C03054=1197.106,-92.383,-39.432,179.291,5.560,149.191
C03055=1197.100,-92.133,-39.443,179.293,5.560,149.190
C03056=1197.095,-91.883,-39.453,179.295,5.561,149.189
C03057=1197.090,-91.634,-39.463,179.298,5.561,149.189
C03058=1197.084,-91.384,-39.474,179.300,5.561,149.188
C03059=1197.080,-91.134,-39.484,179.302,5.561,149.187
C03060=1197.074,-90.885,-39.494,179.305,5.561,149.187
C03061=1197.070,-90.635,-39.505,179.307,5.561,149.186
C03062=1197.064,-90.385,-39.515,179.309,5.561,149.186
C03063=1197.058,-90.136,-39.526,179.311,5.562,149.185
C03064=1197.053,-89.886,-39.536,179.314,5.561,149.184
C03065=1197.048,-89.636,-39.546,179.316,5.562,149.184
C03066=1197.043,-89.386,-39.557,179.318,5.563,149.183
C03067=1197.038,-89.137,-39.566,179.320,5.562,149.182
C03068=1197.032,-88.887,-39.577,179.323,5.563,149.182
C03069=1197.027,-88.637,-39.587,179.325,5.563,149.181
C03070=1197.022,-88.387,-39.597,179.327,5.563,149.180
C03071=1197.017,-88.138,-39.609,179.330,5.563,149.180
C03072=1197.011,-87.888,-39.619,179.332,5.564,149.179
C03073=1197.006,-87.639,-39.629,179.334,5.563,149.178
C03074=1197.001,-87.388,-39.640,179.336,5.564,149.178
C03075=1196.995,-87.139,-39.650,179.339,5.564,149.177
C03076=1196.990,-86.889,-39.661,179.341,5.564,149.177
C03077=1196.985,-86.640,-39.671,179.343,5.564,149.176
C03078=1196.980,-86.389,-39.682,179.345,5.564,149.175
C03079=1196.974,-86.140,-39.692,179.348,5.565,149.175
C03080=1196.969,-85.890,-39.703,179.350,5.564,149.174
C03081=1196.964,-85.640,-39.713,179.352,5.565,149.173
C03082=1196.959,-85.391,-39.723,179.355,5.565,149.172
C03083=1196.954,-85.141,-39.734,179.357,5.565,149.172
C03084=1196.949,-84.892,-39.744,179.359,5.566,149.171
C03085=1196.944,-84.641,-39.755,179.361,5.565,149.171
C03086=1196.938,-84.392,-39.765,179.364,5.566,149.170
C03087=1196.933,-84.142,-39.776,179.366,5.566,149.169
C03088=1196.928,-83.893,-39.786,179.368,5.566,149.169
C03089=1196.923,-83.642,-39.797,179.371,5.567,149.168
C03090=1196.917,-83.393,-39.807,179.373,5.567,149.167
C03091=1196.912,-83.143,-39.818,179.375,5.567,149.167
C03092=1196.907,-82.894,-39.829,179.377,5.567,149.166
C03093=1196.902,-82.643,-39.839,179.380,5.567,149.165
C03094=1196.897,-82.395,-39.850,179.382,5.567,149.165
C03095=1196.892,-82.144,-39.861,179.384,5.567,149.164
C03096=1196.885,-81.894,-39.872,179.387,5.568,149.163
C03097=1196.880,-81.644,-39.882,179.389,5.568,149.163
C03098=1196.875,-81.395,-39.893,179.391,5.568,149.162
C03099=1196.870,-81.145,-39.904,179.393,5.568,149.162
C03100=1196.864,-80.895,-39.914,179.396,5.568,149.161
C03101=1196.860,-80.646,-39.925,179.399,5.569,149.160
C03102=1196.854,-80.396,-39.935,179.400,5.569,149.160
C03103=1196.849,-80.146,-39.946,179.403,5.569,149.159
C03104=1196.844,-79.897,-39.957,179.405,5.569,149.158
C03105=1196.839,-79.647,-39.967,179.407,5.570,149.158
C03106=1196.833,-79.398,-39.978,179.410,5.570,149.157
C03107=1196.828,-79.148,-39.989,179.412,5.570,149.156
C03108=1196.823,-78.898,-39.999,179.415,5.570,149.156
C03109=1196.817,-78.648,-40.011,179.416,5.570,149.155
C03110=1196.812,-78.398,-40.022,179.419,5.571,149.154
C03111=1196.807,-78.149,-40.033,179.421,5.570,149.154
C03112=1196.802,-77.899,-40.043,179.424,5.571,149.153
C03113=1196.797,-77.649,-40.053,179.426,5.571,149.153
C03114=1196.792,-77.400,-40.065,179.428,5.571,149.152
C03115=1196.786,-77.150,-40.075,179.431,5.571,149.151
C03116=1196.782,-76.901,-40.086,179.433,5.571,149.150
C03117=1196.775,-76.651,-40.097,179.435,5.572,149.150
C03118=1196.770,-76.401,-40.108,179.438,5.572,149.149
C03119=1196.765,-76.151,-40.119,179.440,5.572,149.149
C03120=1196.760,-75.902,-40.130,179.442,5.572,149.148
C03121=1196.754,-75.630,-40.141,179.445,5.573,149.147
C03122=1196.748,-75.360,-40.153,179.447,5.572,149.146
C03123=1196.743,-75.089,-40.165,179.450,5.573,149.146
C03124=1196.738,-74.818,-40.177,179.452,5.573,149.145
C03125=1196.732,-74.569,-40.187,179.454,5.573,149.144
C03126=1196.727,-74.319,-40.199,179.457,5.574,149.144
C03127=1196.721,-74.069,-40.209,179.459,5.574,149.143
C03128=1196.716,-73.820,-40.221,179.461,5.574,149.142
C03129=1196.711,-73.569,-40.231,179.464,5.575,149.142
C03130=1196.706,-73.321,-40.242,179.466,5.574,149.141
C03131=1196.701,-73.070,-40.253,179.468,5.575,149.140
C03132=1196.696,-72.820,-40.265,179.471,5.575,149.140
C03133=1196.690,-72.571,-40.275,179.473,5.575,149.139
C03134=1196.685,-72.321,-40.286,179.475,5.575,149.139
C03135=1196.680,-72.072,-40.297,179.477,5.575,149.138
C03136=1196.674,-71.822,-40.308,179.480,5.576,149.137
C03137=1196.670,-71.572,-40.319,179.482,5.576,149.137
C03138=1196.664,-71.323,-40.330,179.484,5.576,149.136
C03139=1196.658,-71.073,-40.342,179.487,5.576,149.135
C03140=1196.654,-70.823,-40.353,179.490,5.577,149.135
C03141=1196.648,-70.573,-40.363,179.491,5.577,149.134
C03142=1196.644,-70.324,-40.374,179.494,5.577,149.133
C03143=1196.638,-70.074,-40.386,179.496,5.577,149.133
C03144=1196.632,-69.824,-40.396,179.499,5.577,149.132
C03145=1196.628,-69.575,-40.408,179.501,5.578,149.131
C03146=1196.622,-69.324,-40.419,179.503,5.578,149.131
C03147=1196.617,-69.075,-40.430,179.506,5.578,149.130
C03148=1196.612,-68.826,-40.441,179.508,5.579,149.129
C03149=1196.607,-68.575,-40.452,179.510,5.578,149.129
C03150=1196.601,-68.326,-40.463,179.513,5.579,149.128
C03151=1196.596,-68.076,-40.474,179.515,5.579,149.127
C03152=1196.592,-67.827,-40.486,179.517,5.579,149.127
C03153=1196.585,-67.577,-40.497,179.520,5.580,149.126
C03154=1196.581,-67.327,-40.508,179.522,5.580,149.126
C03155=1196.576,-67.078,-40.519,179.524,5.580,149.125
C03156=1196.570,-66.828,-40.530,179.527,5.580,149.124
C03157=1196.565,-66.578,-40.541,179.529,5.580,149.123
C03158=1196.560,-66.329,-40.553,179.532,5.581,149.123
C03159=1196.555,-66.079,-40.564,179.533,5.581,149.122
C03160=1196.549,-65.829,-40.575,179.536,5.581,149.122
C03161=1196.544,-65.579,-40.587,179.539,5.581,149.121
C03162=1196.539,-65.330,-40.598,179.541,5.581,149.120
C03163=1196.534,-65.081,-40.609,179.543,5.582,149.120
C03164=1196.528,-64.830,-40.620,179.546,5.582,149.119
C03165=1196.523,-64.580,-40.631,179.548,5.582,149.118
C03166=1196.518,-64.331,-40.643,179.550,5.582,149.118
C03167=1196.513,-64.082,-40.654,179.553,5.583,149.117
C03168=1196.508,-63.832,-40.665,179.555,5.583,149.116
C03169=1196.503,-63.582,-40.677,179.557,5.583,149.116
C03170=1196.498,-63.332,-40.688,179.559,5.583,149.115
C03171=1196.491,-63.083,-40.699,179.562,5.583,149.114
C03172=1196.487,-62.833,-40.711,179.564,5.584,149.114
C03173=1196.482,-62.583,-40.722,179.566,5.584,149.113
C03174=1196.477,-62.333,-40.734,179.569,5.584,149.112
C03175=1196.471,-62.084,-40.745,179.572,5.585,149.112
C03176=1196.466,-61.834,-40.756,179.573,5.585,149.111
C03177=1196.461,-61.584,-40.767,179.576,5.585,149.110
C03178=1196.456,-61.334,-40.779,179.579,5.586,149.110
C03179=1196.451,-61.085,-40.790,179.581,5.585,149.109
C03180=1196.445,-60.835,-40.802,179.583,5.586,149.108
C03181=1196.440,-60.586,-40.813,179.585,5.586,149.108
C03182=1196.435,-60.336,-40.825,179.588,5.586,149.107
C03183=1196.430,-60.086,-40.836,179.590,5.587,149.106
C03184=1196.425,-59.836,-40.848,179.593,5.587,149.106
C03185=1196.419,-59.587,-40.859,179.594,5.587,149.105
C03186=1196.414,-59.337,-40.871,179.597,5.587,149.105
C03187=1196.409,-59.088,-40.882,179.600,5.588,149.104
C03188=1196.404,-58.838,-40.894,179.602,5.587,149.103
C03189=1196.399,-58.588,-40.905,179.605,5.588,149.102
C03190=1196.393,-58.338,-40.916,179.607,5.589,149.102
C03191=1196.388,-58.089,-40.928,179.609,5.588,149.101
C03192=1196.383,-57.839,-40.939,179.612,5.589,149.101
C03193=1196.378,-57.589,-40.951,179.614,5.588,149.100
C03194=1196.372,-57.339,-40.963,179.616,5.589,149.099
C03195=1196.368,-57.090,-40.974,179.618,5.590,149.099
C03196=1196.362,-56.840,-40.985,179.621,5.589,149.098
C03197=1196.357,-56.591,-40.997,179.623,5.590,149.097
C03198=1196.352,-56.342,-41.009,179.626,5.590,149.097
C03199=1196.347,-56.092,-41.021,179.627,5.590,149.096
C03200=1196.342,-55.842,-41.032,179.630,5.591,149.095
C03201=1196.336,-55.592,-41.044,179.633,5.591,149.095
C03202=1196.332,-55.342,-41.056,179.635,5.591,149.094
C03203=1196.326,-55.092,-41.068,179.638,5.591,149.093
C03204=1196.321,-54.844,-41.078,179.640,5.592,149.093
C03205=1196.316,-54.594,-41.090,179.642,5.592,149.092
C03206=1196.310,-54.344,-41.102,179.644,5.592,149.091
C03207=1196.305,-54.094,-41.114,179.647,5.593,149.091
C03208=1196.300,-53.844,-41.125,179.650,5.593,149.090
C03209=1196.295,-53.594,-41.137,179.651,5.593,149.090
C03210=1196.290,-53.345,-41.149,179.654,5.593,149.089
C03211=1196.285,-53.095,-41.161,179.657,5.594,149.088
C03212=1196.280,-52.846,-41.172,179.659,5.594,149.087
C03213=1196.274,-52.596,-41.184,179.661,5.594,149.087
C03214=1196.269,-52.347,-41.195,179.664,5.595,149.086
C03215=1196.264,-52.097,-41.207,179.666,5.594,149.086
C03216=1196.258,-51.847,-41.219,179.668,5.595,149.085
C03217=1196.254,-51.598,-41.231,179.671,5.595,149.084
C03218=1196.249,-51.348,-41.243,179.673,5.595,149.083
C03219=1196.243,-51.098,-41.255,179.675,5.596,149.083
C03220=1196.239,-50.848,-41.266,179.678,5.596,149.082
C03221=1196.233,-50.598,-41.278,179.680,5.596,149.082
C03222=1196.228,-50.349,-41.291,179.683,5.596,149.081
C03223=1196.223,-50.099,-41.302,179.685,5.597,149.080
C03224=1196.218,-49.850,-41.314,179.687,5.597,149.080
C03225=1196.212,-49.580,-41.326,179.690,5.597,149.079
C03226=1196.207,-49.310,-41.339,179.692,5.598,149.078
C03227=1196.201,-49.039,-41.352,179.695,5.598,149.078
C03228=1196.195,-48.769,-41.365,179.698,5.599,149.077
C03229=1196.190,-48.520,-41.377,179.700,5.599,149.076
C03230=1196.185,-48.270,-41.389,179.702,5.599,149.075
C03231=1196.179,-48.020,-41.401,179.705,5.599,149.075
C03232=1196.174,-47.770,-41.413,179.708,5.600,149.074
C03233=1196.169,-47.521,-41.424,179.709,5.600,149.074
C03234=1196.164,-47.271,-41.436,179.712,5.600,149.073
C03235=1196.159,-47.022,-41.449,179.715,5.601,149.072
C03236=1196.153,-46.772,-41.461,179.717,5.600,149.071
C03237=1196.149,-46.522,-41.472,179.719,5.601,149.071
C03238=1196.143,-46.273,-41.485,179.722,5.601,149.070
C03239=1196.138,-46.023,-41.497,179.724,5.602,149.070
C03240=1196.133,-45.773,-41.508,179.726,5.602,149.069
C03241=1196.128,-45.524,-41.520,179.729,5.602,149.068
C03242=1196.123,-45.274,-41.532,179.732,5.602,149.067
C03243=1196.117,-45.024,-41.544,179.733,5.602,149.067
C03244=1196.112,-44.775,-41.557,179.736,5.603,149.066
C03245=1196.107,-44.525,-41.569,179.739,5.603,149.066
C03246=1196.102,-44.275,-41.581,179.741,5.603,149.065
C03247=1196.097,-44.026,-41.593,179.743,5.603,149.064
C03248=1196.092,-43.776,-41.605,179.746,5.604,149.064
C03249=1196.086,-43.526,-41.617,179.748,5.605,149.063
C03250=1196.081,-43.276,-41.629,179.750,5.604,149.062
C03251=1196.076,-43.027,-41.642,179.753,5.605,149.062
C03252=1196.070,-42.777,-41.653,179.756,5.605,149.061
C03253=1196.066,-42.528,-41.665,179.758,5.606,149.060
C03254=1196.061,-42.278,-41.677,179.760,5.606,149.060
C03255=1196.055,-42.028,-41.689,179.763,5.606,149.059
C03256=1196.050,-41.779,-41.702,179.765,5.607,149.058
C03257=1196.045,-41.529,-41.714,179.767,5.606,149.058
C03258=1196.040,-41.280,-41.726,179.769,5.607,149.057
C03259=1196.035,-41.029,-41.739,179.772,5.608,149.056
C03260=1196.030,-40.780,-41.751,179.775,5.608,149.056
C03261=1196.025,-40.530,-41.762,179.777,5.608,149.055
C03262=1196.020,-40.281,-41.775,179.779,5.608,149.054
C03263=1196.014,-40.031,-41.787,179.782,5.609,149.054
C03264=1196.009,-39.782,-41.800,179.784,5.609,149.053
C03265=1196.004,-39.532,-41.811,179.786,5.609,149.053
C03266=1195.999,-39.282,-41.824,179.789,5.610,149.052
C03267=1195.993,-39.032,-41.836,179.792,5.610,149.051
C03268=1195.988,-38.783,-41.849,179.793,5.610,149.051
C03269=1195.983,-38.533,-41.860,179.796,5.610,149.050
C03270=1195.978,-38.284,-41.873,179.799,5.611,149.049
C03271=1195.973,-38.034,-41.886,179.801,5.611,149.049
C03272=1195.968,-37.784,-41.898,179.803,5.611,149.048
C03273=1195.963,-37.535,-41.910,179.806,5.612,149.047
C03274=1195.957,-37.285,-41.922,179.808,5.612,149.047
C03275=1195.952,-37.035,-41.935,179.811,5.613,149.046
C03276=1195.947,-36.786,-41.948,179.813,5.612,149.045
C03277=1195.941,-36.536,-41.959,179.816,5.613,149.045
C03278=1195.936,-36.287,-41.972,179.818,5.614,149.044
C03279=1195.931,-36.036,-41.984,179.820,5.614,149.043
C03280=1195.926,-35.787,-41.997,179.823,5.614,149.043
C03281=1195.921,-35.538,-42.010,179.825,5.614,149.042
C03282=1195.916,-35.288,-42.021,179.828,5.615,149.041
C03283=1195.911,-35.038,-42.034,179.830,5.616,149.041
C03284=1195.906,-34.789,-42.047,179.832,5.615,149.040
C03285=1195.900,-34.539,-42.058,179.835,5.616,149.039
C03286=1195.896,-34.289,-42.071,179.837,5.616,149.039
C03287=1195.890,-34.040,-42.084,179.840,5.617,149.038
C03288=1195.885,-33.790,-42.096,179.842,5.616,149.037
C03289=1195.880,-33.540,-42.109,179.844,5.617,149.037
C03290=1195.875,-33.291,-42.121,179.847,5.618,149.036
C03291=1195.870,-33.042,-42.134,179.850,5.618,149.035
C03292=1195.865,-32.791,-42.146,179.852,5.618,149.035
C03293=1195.860,-32.542,-42.159,179.854,5.618,149.034
C03294=1195.855,-32.293,-42.171,179.857,5.619,149.034
C03295=1195.849,-32.043,-42.184,179.859,5.619,149.033
C03296=1195.844,-31.793,-42.196,179.861,5.619,149.032
C03297=1195.839,-31.543,-42.209,179.864,5.620,149.032
C03298=1195.834,-31.294,-42.222,179.867,5.620,149.031
C03299=1195.829,-31.044,-42.234,179.869,5.621,149.030
C03300=1195.823,-30.794,-42.246,179.871,5.621,149.030
C03301=1195.818,-30.545,-42.259,179.874,5.621,149.029
C03302=1195.813,-30.295,-42.272,179.876,5.621,149.028
C03303=1195.808,-30.046,-42.284,179.879,5.622,149.028
C03304=1195.803,-29.796,-42.297,179.881,5.622,149.027
C03305=1195.798,-29.547,-42.310,179.883,5.622,149.026
C03306=1195.792,-29.296,-42.323,179.886,5.623,149.026
C03307=1195.787,-29.047,-42.335,179.888,5.623,149.025
C03308=1195.782,-28.797,-42.348,179.891,5.624,149.024
C03309=1195.777,-28.548,-42.360,179.893,5.624,149.024
C03310=1195.773,-28.298,-42.373,179.895,5.624,149.023
C03311=1195.767,-28.049,-42.386,179.898,5.625,149.022
C03312=1195.762,-27.800,-42.399,179.901,5.625,149.022
C03313=1195.756,-27.549,-42.411,179.903,5.625,149.021
C03314=1195.752,-27.299,-42.424,179.905,5.625,149.020
C03315=1195.747,-27.050,-42.437,179.908,5.626,149.020
C03316=1195.741,-26.801,-42.449,179.910,5.627,149.019
C03317=1195.736,-26.551,-42.462,179.913,5.627,149.018
C03318=1195.731,-26.301,-42.475,179.915,5.627,149.018
C03319=1195.726,-26.052,-42.488,179.918,5.627,149.017
C03320=1195.721,-25.802,-42.501,179.920,5.628,149.017
C03321=1195.716,-25.552,-42.513,179.923,5.629,149.016
C03322=1195.711,-25.303,-42.526,179.925,5.629,149.015
C03323=1195.705,-25.053,-42.539,179.927,5.629,149.015
C03324=1195.700,-24.804,-42.552,179.930,5.629,149.014
C03325=1195.696,-24.554,-42.565,179.932,5.630,149.013
C03326=1195.691,-24.305,-42.577,179.935,5.630,149.013
C03327=1195.685,-24.055,-42.591,179.937,5.631,149.012
C03328=1195.680,-23.805,-42.604,179.939,5.631,149.011
C03329=1195.675,-23.536,-42.617,179.942,5.631,149.011
C03330=1195.669,-23.266,-42.631,179.945,5.632,149.010
C03331=1195.664,-22.996,-42.645,179.947,5.632,149.009
C03332=1195.657,-22.727,-42.659,179.950,5.632,149.008
C03333=1195.653,-22.477,-42.672,179.953,5.633,149.008
C03334=1195.647,-22.227,-42.685,179.955,5.633,149.007
C03335=1195.642,-21.978,-42.698,179.957,5.633,149.007
C03336=1195.637,-21.728,-42.711,179.960,5.634,149.006
C03337=1195.632,-21.479,-42.723,179.962,5.634,149.005
C03338=1195.627,-21.230,-42.737,179.965,5.635,149.005
C03339=1195.622,-20.980,-42.750,179.968,5.635,149.004
C03340=1195.617,-20.730,-42.763,179.970,5.636,149.003
C03341=1195.612,-20.480,-42.776,179.972,5.636,149.003
C03342=1195.607,-20.231,-42.789,179.975,5.636,149.002
C03343=1195.602,-19.981,-42.801,179.977,5.637,149.001
C03344=1195.596,-19.731,-42.815,179.980,5.637,149.001
C03345=1195.591,-19.482,-42.828,179.982,5.638,149.000
C03346=1195.586,-19.233,-42.841,179.984,5.638,148.999
C03347=1195.581,-18.983,-42.854,179.987,5.638,148.999
C03348=1195.576,-18.733,-42.867,179.989,5.639,148.998
C03349=1195.571,-18.483,-42.881,179.992,5.639,148.997
C03350=1195.566,-18.234,-42.893,179.995,5.640,148.997
C03351=1195.560,-17.984,-42.906,179.996,5.640,148.996
C03352=1195.556,-17.735,-42.920,179.999,5.640,148.995
C03353=1195.550,-17.485,-42.933,-179.998,5.641,148.995
C03354=1195.545,-17.235,-42.946,-179.996,5.641,148.994
C03355=1195.540,-16.986,-42.959,-179.993,5.642,148.993
C03356=1195.534,-16.736,-42.972,-179.991,5.642,148.993
C03357=1195.530,-16.487,-42.986,-179.989,5.642,148.992
C03358=1195.525,-16.237,-42.998,-179.986,5.643,148.992
C03359=1195.520,-15.987,-43.012,-179.983,5.643,148.991
C03360=1195.514,-15.738,-43.024,-179.981,5.643,148.990
C03361=1195.509,-15.488,-43.039,-179.979,5.644,148.990
C03362=1195.504,-15.239,-43.051,-179.976,5.645,148.989
C03363=1195.498,-14.989,-43.065,-179.974,5.644,148.988
C03364=1195.494,-14.739,-43.077,-179.971,5.645,148.988
C03365=1195.488,-14.490,-43.091,-179.969,5.645,148.987
C03366=1195.484,-14.240,-43.104,-179.966,5.646,148.986
C03367=1195.479,-13.991,-43.117,-179.964,5.647,148.986
C03368=1195.474,-13.741,-43.131,-179.961,5.647,148.985
C03369=1195.469,-13.492,-43.144,-179.959,5.647,148.984
C03370=1195.463,-13.241,-43.157,-179.956,5.647,148.984
C03371=1195.459,-12.993,-43.171,-179.954,5.648,148.983
C03372=1195.453,-12.742,-43.184,-179.952,5.649,148.983
C03373=1195.448,-12.493,-43.197,-179.949,5.649,148.982
C03374=1195.443,-12.243,-43.211,-179.946,5.650,148.981
C03375=1195.437,-11.994,-43.224,-179.944,5.649,148.980
C03376=1195.433,-11.744,-43.238,-179.942,5.650,148.980
C03377=1195.427,-11.495,-43.251,-179.939,5.651,148.979
C03378=1195.423,-11.245,-43.264,-179.937,5.651,148.979
C03379=1195.417,-10.996,-43.278,-179.934,5.652,148.978
C03380=1195.413,-10.746,-43.291,-179.931,5.652,148.977
C03381=1195.407,-10.497,-43.305,-179.929,5.653,148.977
C03382=1195.403,-10.247,-43.318,-179.927,5.653,148.976
C03383=1195.397,-9.997,-43.331,-179.924,5.653,148.975
C03384=1195.393,-9.747,-43.345,-179.922,5.654,148.975
C03385=1195.387,-9.498,-43.358,-179.919,5.654,148.974
C03386=1195.382,-9.248,-43.372,-179.917,5.655,148.974
C03387=1195.377,-8.999,-43.385,-179.914,5.655,148.973
C03388=1195.372,-8.749,-43.399,-179.912,5.656,148.972
C03389=1195.367,-8.500,-43.412,-179.910,5.656,148.971
C03390=1195.362,-8.250,-43.426,-179.907,5.656,148.971
C03391=1195.356,-8.000,-43.439,-179.905,5.657,148.970
C03392=1195.352,-7.751,-43.453,-179.902,5.657,148.970
C03393=1195.346,-7.501,-43.467,-179.899,5.658,148.969
C03394=1195.341,-7.252,-43.480,-179.897,5.658,148.968
C03395=1195.336,-7.002,-43.493,-179.894,5.659,148.968
C03396=1195.331,-6.753,-43.507,-179.892,5.660,148.967
C03397=1195.326,-6.503,-43.520,-179.890,5.659,148.966
C03398=1195.321,-6.254,-43.534,-179.887,5.660,148.966
C03399=1195.316,-6.004,-43.548,-179.885,5.660,148.965
C03400=1195.311,-5.754,-43.561,-179.882,5.661,148.964
C03401=1195.306,-5.505,-43.575,-179.880,5.662,148.964
C03402=1195.300,-5.255,-43.589,-179.877,5.662,148.963
C03403=1195.295,-5.006,-43.602,-179.874,5.663,148.962
C03404=1195.290,-4.756,-43.616,-179.872,5.663,148.962
C03405=1195.285,-4.507,-43.630,-179.870,5.663,148.961
C03406=1195.280,-4.257,-43.643,-179.868,5.664,148.961
C03407=1195.275,-4.007,-43.657,-179.865,5.664,148.960
C03408=1195.270,-3.758,-43.671,-179.862,5.665,148.959
C03409=1195.265,-3.508,-43.685,-179.860,5.665,148.959
C03410=1195.260,-3.258,-43.698,-179.857,5.665,148.958
C03411=1195.255,-3.009,-43.712,-179.855,5.666,148.957
C03412=1195.250,-2.759,-43.726,-179.852,5.667,148.957
C03413=1195.244,-2.510,-43.739,-179.849,5.667,148.956
C03414=1195.240,-2.260,-43.753,-179.847,5.667,148.955
C03415=1195.235,-2.011,-43.767,-179.845,5.667,148.955
C03416=1195.229,-1.761,-43.781,-179.843,5.668,148.954
C03417=1195.224,-1.512,-43.794,-179.840,5.669,148.953
C03418=1195.220,-1.262,-43.809,-179.837,5.669,148.953
C03419=1195.214,-1.013,-43.822,-179.835,5.670,148.952
C03420=1195.209,-0.763,-43.836,-179.832,5.670,148.951
C03421=1195.204,-0.513,-43.850,-179.830,5.671,148.951
C03422=1195.199,-0.264,-43.864,-179.827,5.672,148.950
C03423=1195.194,-0.014,-43.878,-179.825,5.671,148.950
C03424=1195.189,0.236,-43.891,-179.822,5.672,148.949
C03425=1195.183,0.485,-43.905,-179.820,5.672,148.948
C03426=1195.178,0.735,-43.920,-179.818,5.673,148.948
C03427=1195.174,0.984,-43.933,-179.815,5.674,148.947
C03428=1195.168,1.234,-43.947,-179.812,5.674,148.946
C03429=1195.163,1.483,-43.961,-179.810,5.675,148.946
C03430=1195.158,1.733,-43.975,-179.807,5.675,148.945
C03431=1195.153,1.982,-43.989,-179.805,5.676,148.945
C03432=1195.148,2.232,-44.003,-179.802,5.676,148.944
C03433=1195.142,2.501,-44.018,-179.799,5.677,148.943
C03434=1195.137,2.771,-44.033,-179.797,5.677,148.942
C03435=1195.131,3.039,-44.048,-179.794,5.678,148.942
C03436=1195.126,3.308,-44.064,-179.792,5.678,148.941
C03437=1195.121,3.558,-44.077,-179.789,5.679,148.940
C03438=1195.116,3.808,-44.091,-179.786,5.679,148.940
C03439=1195.111,4.057,-44.105,-179.784,5.680,148.939
C03440=1195.106,4.307,-44.119,-179.781,5.681,148.939
C03441=1195.101,4.556,-44.133,-179.779,5.681,148.938
C03442=1195.096,4.806,-44.148,-179.777,5.681,148.937
C03443=1195.090,5.055,-44.162,-179.774,5.681,148.937
C03444=1195.085,5.305,-44.176,-179.772,5.682,148.936
C03445=1195.080,5.554,-44.190,-179.769,5.683,148.935
C03446=1195.075,5.804,-44.204,-179.767,5.683,148.935
C03447=1195.071,6.053,-44.218,-179.764,5.684,148.934
C03448=1195.066,6.303,-44.232,-179.761,5.684,148.933
C03449=1195.061,6.552,-44.246,-179.759,5.685,148.933
C03450=1195.056,6.802,-44.260,-179.756,5.686,148.932
C03451=1195.051,7.052,-44.275,-179.754,5.686,148.931
C03452=1195.045,7.301,-44.289,-179.751,5.687,148.931
C03453=1195.040,7.550,-44.303,-179.749,5.687,148.930
C03454=1195.035,7.800,-44.317,-179.746,5.688,148.930
C03455=1195.030,8.050,-44.332,-179.744,5.688,148.929
C03456=1195.025,8.299,-44.345,-179.741,5.689,148.928
C03457=1195.020,8.549,-44.360,-179.739,5.689,148.928
C03458=1195.015,8.798,-44.374,-179.737,5.689,148.927
C03459=1195.010,9.048,-44.388,-179.734,5.690,148.926
C03460=1195.005,9.298,-44.403,-179.731,5.690,148.926
C03461=1195.000,9.547,-44.417,-179.729,5.691,148.925
C03462=1194.994,9.796,-44.431,-179.727,5.692,148.925
C03463=1194.989,10.046,-44.445,-179.724,5.692,148.924
C03464=1194.985,10.296,-44.459,-179.721,5.693,148.923
C03465=1194.980,10.546,-44.474,-179.719,5.693,148.923
C03466=1194.975,10.795,-44.488,-179.716,5.694,148.922
C03467=1194.969,11.044,-44.502,-179.714,5.695,148.921
C03468=1194.964,11.293,-44.517,-179.711,5.695,148.921
C03469=1194.959,11.543,-44.531,-179.709,5.696,148.920
C03470=1194.954,11.793,-44.545,-179.706,5.696,148.919
C03471=1194.949,12.043,-44.560,-179.704,5.697,148.919
C03472=1194.944,12.292,-44.574,-179.701,5.697,148.918
C03473=1194.939,12.542,-44.589,-179.698,5.698,148.918
C03474=1194.934,12.791,-44.603,-179.696,5.698,148.917
C03475=1194.929,13.040,-44.618,-179.693,5.699,148.916
C03476=1194.924,13.290,-44.632,-179.691,5.700,148.916
C03477=1194.919,13.540,-44.646,-179.688,5.700,148.915
C03478=1194.914,13.789,-44.660,-179.686,5.701,148.914
C03479=1194.909,14.039,-44.675,-179.683,5.701,148.914
C03480=1194.904,14.288,-44.690,-179.681,5.701,148.913
C03481=1194.899,14.538,-44.705,-179.679,5.702,148.913
C03482=1194.893,14.787,-44.719,-179.676,5.702,148.912
C03483=1194.888,15.036,-44.733,-179.674,5.703,148.911
C03484=1194.883,15.286,-44.748,-179.671,5.704,148.911
C03485=1194.878,15.536,-44.762,-179.669,5.704,148.910
C03486=1194.873,15.785,-44.776,-179.666,5.705,148.909
C03487=1194.868,16.035,-44.792,-179.663,5.705,148.909
C03488=1194.863,16.285,-44.806,-179.661,5.706,148.908
C03489=1194.858,16.534,-44.820,-179.659,5.707,148.908
C03490=1194.854,16.783,-44.835,-179.656,5.707,148.907
C03491=1194.849,17.033,-44.850,-179.653,5.708,148.906
C03492=1194.844,17.283,-44.864,-179.651,5.708,148.905
C03493=1194.838,17.532,-44.880,-179.649,5.709,148.905
C03494=1194.833,17.782,-44.894,-179.646,5.709,148.904
C03495=1194.828,18.031,-44.908,-179.643,5.710,148.904
C03496=1194.823,18.280,-44.923,-179.641,5.710,148.903
C03497=1194.818,18.530,-44.937,-179.638,5.711,148.903
C03498=1194.812,18.780,-44.952,-179.636,5.712,148.902
C03499=1194.808,19.029,-44.967,-179.633,5.712,148.901
C03500=1194.803,19.279,-44.981,-179.630,5.713,148.900
C03501=1194.798,19.528,-44.995,-179.628,5.714,148.900
C03502=1194.792,19.778,-45.011,-179.626,5.714,148.899
C03503=1194.787,20.027,-45.025,-179.623,5.715,148.899
C03504=1194.783,20.276,-45.040,-179.620,5.715,148.898
C03505=1194.778,20.526,-45.055,-179.618,5.716,148.897
C03506=1194.773,20.776,-45.070,-179.616,5.717,148.897
C03507=1194.768,21.025,-45.084,-179.613,5.717,148.896
C03508=1194.763,21.274,-45.099,-179.610,5.718,148.895
C03509=1194.757,21.524,-45.114,-179.608,5.718,148.895
C03510=1194.752,21.774,-45.129,-179.605,5.719,148.894
C03511=1194.748,22.023,-45.144,-179.603,5.720,148.894
C03512=1194.742,22.273,-45.158,-179.600,5.720,148.893
C03513=1194.737,22.522,-45.173,-179.597,5.721,148.892
C03514=1194.732,22.772,-45.188,-179.595,5.721,148.892
C03515=1194.727,23.021,-45.203,-179.593,5.722,148.891
C03516=1194.722,23.271,-45.218,-179.590,5.722,148.891
C03517=1194.717,23.520,-45.233,-179.587,5.723,148.890
C03518=1194.712,23.770,-45.248,-179.585,5.724,148.889
C03519=1194.707,24.019,-45.262,-179.583,5.724,148.889
C03520=1194.702,24.268,-45.277,-179.580,5.725,148.888
C03521=1194.697,24.518,-45.292,-179.577,5.725,148.887
C03522=1194.692,24.768,-45.307,-179.575,5.726,148.887
C03523=1194.687,25.017,-45.322,-179.572,5.727,148.886
C03524=1194.682,25.267,-45.338,-179.570,5.727,148.886
C03525=1194.678,25.516,-45.353,-179.567,5.728,148.885
C03526=1194.672,25.766,-45.367,-179.565,5.729,148.884
C03527=1194.667,26.016,-45.382,-179.562,5.730,148.884
C03528=1194.662,26.265,-45.397,-179.559,5.730,148.883
C03529=1194.657,26.515,-45.412,-179.557,5.731,148.882
C03530=1194.652,26.764,-45.427,-179.554,5.732,148.882
C03531=1194.647,27.014,-45.442,-179.552,5.732,148.881
C03532=1194.642,27.263,-45.457,-179.549,5.733,148.881
C03533=1194.637,27.512,-45.472,-179.546,5.733,148.880
C03534=1194.632,27.762,-45.487,-179.544,5.734,148.879
C03535=1194.627,28.011,-45.502,-179.542,5.735,148.879
C03536=1194.622,28.260,-45.518,-179.539,5.735,148.878
C03537=1194.617,28.530,-45.534,-179.536,5.736,148.877
C03538=1194.611,28.799,-45.550,-179.534,5.736,148.877
C03539=1194.606,29.067,-45.566,-179.531,5.737,148.876
C03540=1194.600,29.336,-45.583,-179.528,5.738,148.875
C03541=1194.596,29.585,-45.598,-179.526,5.739,148.875
C03542=1194.590,29.835,-45.613,-179.523,5.739,148.874
C03543=1194.585,30.085,-45.628,-179.520,5.740,148.874
C03544=1194.580,30.334,-45.643,-179.518,5.740,148.873
C03545=1194.575,30.583,-45.658,-179.516,5.741,148.872
C03546=1194.570,30.832,-45.674,-179.513,5.742,148.872
C03547=1194.566,31.082,-45.689,-179.510,5.742,148.871
C03548=1194.560,31.332,-45.704,-179.508,5.743,148.871
C03549=1194.555,31.582,-45.720,-179.505,5.744,148.870
C03550=1194.550,31.831,-45.735,-179.503,5.744,148.869
C03551=1194.545,32.080,-45.750,-179.500,5.745,148.869
C03552=1194.540,32.329,-45.765,-179.498,5.746,148.868
C03553=1194.535,32.580,-45.780,-179.495,5.746,148.867
C03554=1194.531,32.829,-45.795,-179.493,5.747,148.867
C03555=1194.525,33.078,-45.811,-179.490,5.748,148.866
C03556=1194.520,33.328,-45.826,-179.487,5.749,148.866
C03557=1194.515,33.577,-45.842,-179.485,5.749,148.865
C03558=1194.510,33.826,-45.857,-179.482,5.750,148.864
C03559=1194.506,34.076,-45.872,-179.480,5.751,148.864
C03560=1194.500,34.326,-45.888,-179.477,5.751,148.863
C03561=1194.495,34.575,-45.902,-179.475,5.752,148.863
C03562=1194.490,34.825,-45.918,-179.472,5.752,148.862
C03563=1194.485,35.074,-45.934,-179.470,5.753,148.861
C03564=1194.480,35.324,-45.949,-179.467,5.754,148.861
C03565=1194.475,35.573,-45.964,-179.465,5.754,148.860
C03566=1194.470,35.823,-45.980,-179.462,5.755,148.859
C03567=1194.465,36.072,-45.995,-179.460,5.756,148.859
C03568=1194.460,36.322,-46.011,-179.457,5.756,148.858
C03569=1194.456,36.571,-46.026,-179.454,5.758,148.858
C03570=1194.450,36.820,-46.042,-179.452,5.758,148.857
C03571=1194.445,37.070,-46.057,-179.449,5.759,148.856
C03572=1194.440,37.319,-46.072,-179.446,5.759,148.856
C03573=1194.435,37.569,-46.088,-179.444,5.760,148.855
C03574=1194.430,37.818,-46.104,-179.442,5.761,148.855
C03575=1194.425,38.068,-46.119,-179.439,5.761,148.854
C03576=1194.420,38.317,-46.134,-179.436,5.762,148.853
C03577=1194.415,38.567,-46.150,-179.434,5.763,148.853
C03578=1194.410,38.816,-46.166,-179.432,5.763,148.852
C03579=1194.405,39.065,-46.181,-179.428,5.765,148.852
C03580=1194.400,39.316,-46.197,-179.426,5.765,148.851
C03581=1194.395,39.565,-46.212,-179.424,5.766,148.850
C03582=1194.390,39.814,-46.229,-179.421,5.767,148.850
C03583=1194.385,40.063,-46.244,-179.418,5.767,148.849
C03584=1194.380,40.313,-46.260,-179.416,5.768,148.849
C03585=1194.375,40.562,-46.275,-179.413,5.768,148.848
C03586=1194.370,40.812,-46.291,-179.411,5.769,148.847
C03587=1194.366,41.062,-46.306,-179.408,5.769,148.847
C03588=1194.360,41.311,-46.322,-179.406,5.770,148.846
C03589=1194.355,41.560,-46.337,-179.403,5.772,148.845
C03590=1194.350,41.810,-46.354,-179.400,5.772,148.845
C03591=1194.346,42.059,-46.369,-179.398,5.773,148.844
C03592=1194.340,42.308,-46.385,-179.395,5.774,148.844
C03593=1194.336,42.558,-46.401,-179.393,5.774,148.843
C03594=1194.330,42.808,-46.416,-179.391,5.775,148.843
C03595=1194.325,43.057,-46.432,-179.388,5.776,148.842
C03596=1194.320,43.307,-46.448,-179.385,5.776,148.841
C03597=1194.316,43.556,-46.463,-179.382,5.777,148.841
C03598=1194.310,43.805,-46.479,-179.380,5.778,148.840
C03599=1194.306,44.055,-46.495,-179.377,5.779,148.839
C03600=1194.300,44.304,-46.511,-179.375,5.779,148.839
C03601=1194.295,44.553,-46.527,-179.373,5.780,148.838
C03602=1194.290,44.804,-46.543,-179.370,5.781,148.838
C03603=1194.286,45.053,-46.558,-179.367,5.781,148.837
C03604=1194.281,45.301,-46.574,-179.365,5.782,148.837
C03605=1194.276,45.552,-46.590,-179.362,5.784,148.836
C03606=1194.270,45.801,-46.606,-179.359,5.784,148.835
C03607=1194.266,46.050,-46.622,-179.357,5.785,148.835
C03608=1194.260,46.300,-46.638,-179.354,5.785,148.834
C03609=1194.255,46.549,-46.653,-179.352,5.786,148.833
C03610=1194.251,46.799,-46.670,-179.349,5.786,148.833
C03611=1194.245,47.048,-46.686,-179.347,5.787,148.832
C03612=1194.241,47.298,-46.701,-179.344,5.789,148.832
C03613=1194.236,47.547,-46.717,-179.341,5.789,148.831
C03614=1194.231,47.796,-46.733,-179.339,5.790,148.831
C03615=1194.226,48.046,-46.749,-179.336,5.791,148.830
C03616=1194.221,48.295,-46.765,-179.334,5.791,148.829
C03617=1194.216,48.545,-46.781,-179.332,5.792,148.829
C03618=1194.211,48.794,-46.797,-179.329,5.793,148.828
C03619=1194.206,49.044,-46.813,-179.326,5.794,148.827
C03620=1194.201,49.293,-46.830,-179.324,5.795,148.827
C03621=1194.196,49.542,-46.845,-179.321,5.795,148.826
C03622=1194.191,49.792,-46.861,-179.318,5.796,148.826
C03623=1194.186,50.041,-46.878,-179.316,5.796,148.825
C03624=1194.181,50.291,-46.893,-179.314,5.797,148.825
C03625=1194.176,50.540,-46.910,-179.311,5.798,148.824
C03626=1194.171,50.790,-46.926,-179.308,5.799,148.823
C03627=1194.166,51.039,-46.942,-179.305,5.800,148.823
C03628=1194.161,51.289,-46.958,-179.303,5.801,148.822
C03629=1194.156,51.538,-46.974,-179.300,5.801,148.821
C03630=1194.151,51.788,-46.990,-179.298,5.802,148.821
C03631=1194.146,52.037,-47.007,-179.295,5.803,148.820
C03632=1194.142,52.287,-47.023,-179.292,5.804,148.820
C03633=1194.137,52.536,-47.039,-179.290,5.805,148.819
C03634=1194.132,52.786,-47.055,-179.287,5.805,148.819
C03635=1194.127,53.034,-47.071,-179.285,5.806,148.818
C03636=1194.122,53.284,-47.088,-179.283,5.807,148.817
C03637=1194.117,53.533,-47.103,-179.279,5.808,148.817
C03638=1194.112,53.783,-47.120,-179.277,5.809,148.816
C03639=1194.107,54.032,-47.136,-179.275,5.810,148.816
C03640=1194.102,54.282,-47.152,-179.272,5.810,148.815
C03641=1194.096,54.550,-47.170,-179.269,5.811,148.814
C03642=1194.091,54.818,-47.188,-179.266,5.812,148.814
C03643=1194.086,55.087,-47.205,-179.264,5.812,148.813
C03644=1194.081,55.355,-47.223,-179.261,5.813,148.813
C03645=1194.076,55.605,-47.239,-179.258,5.815,148.812
C03646=1194.071,55.854,-47.255,-179.256,5.815,148.811
C03647=1194.065,56.105,-47.272,-179.253,5.816,148.811
C03648=1194.060,56.353,-47.288,-179.251,5.817,148.810
C03649=1194.056,56.603,-47.305,-179.248,5.817,148.809
C03650=1194.051,56.852,-47.321,-179.245,5.819,148.809
C03651=1194.046,57.102,-47.337,-179.243,5.819,148.808
C03652=1194.041,57.351,-47.353,-179.240,5.820,148.808
C03653=1194.036,57.600,-47.370,-179.238,5.821,148.807
